LIN {X 0,Y 368.058,Z 315.59,A -85,B 0,C 180,E1 -13017.849,E2 -13017.849} C_VEL
LIN {X 0,Y 375.549,Z 331.898,A -85,B 0,C 180,E1 -13019.02,E2 -13019.02} C_VEL
LIN {X 0,Y 376.727,Z 335.393,A -85,B 0,C 180,E1 -13019.219,E2 -13019.219} C_VEL
LIN {X 0,Y 381.091,Z 359.299,A -85,B 0,C 180,E1 -13020.193,E2 -13020.193} C_VEL
LIN {X 0,Y 377.486,Z 482.299,A -85,B 0,C 180,E1 -13022.675,E2 -13022.675} C_VEL
LIN {X 0,Y 376.481,Z 498.143,A -85,B 0,C 180,E1 -13023.197,E2 -13023.197} C_VEL
LIN {X 0,Y 375.186,Z 512.324,A -85,B 0,C 180,E1 -13023.862,E2 -13023.862} C_VEL
LIN {X 0,Y 373.616,Z 526.793,A -85,B 0,C 180,E1 -13024.762,E2 -13024.762} C_VEL
LIN {X 0,Y 371.852,Z 540.842,A -85,B 0,C 180,E1 -13025.877,E2 -13025.877} C_VEL
LIN {X 0,Y 369.933,Z 554.519,A -85,B 0,C 180,E1 -13027.228,E2 -13027.228} C_VEL
LIN {X 0,Y 367.984,Z 566.938,A -85,B 0,C 180,E1 -13028.724,E2 -13028.724} C_VEL
LIN {X 0,Y 366.187,Z 578.952,A -85,B 0,C 180,E1 -13030.485,E2 -13030.485} C_VEL
LIN {X 0,Y 364.472,Z 589.352,A -85,B 0,C 180,E1 -13032.321,E2 -13032.321} C_VEL
LIN {X 0,Y 363.116,Z 598.534,A -85,B 0,C 180,E1 -13034.279,E2 -13034.279} C_VEL
LIN {X 0,Y 361.947,Z 607.188,A -85,B 0,C 180,E1 -13036.527,E2 -13036.527} C_VEL
LIN {X 0,Y 361.137,Z 614.142,A -85,B 0,C 180,E1 -13038.779,E2 -13038.779} C_VEL
LIN {X 0,Y 360.63,Z 619.607,A -85,B 0,C 180,E1 -13041.031,E2 -13041.031} C_VEL
LIN {X 0,Y 360.378,Z 623.728,A -85,B 0,C 180,E1 -13043.281,E2 -13043.281} C_VEL
LIN {X 0,Y 360.294,Z 626.602,A -85,B 0,C 180,E1 -13045.525,E2 -13045.525} C_VEL
LIN {X 0,Y 360.257,Z 628.286,A -85,B 0,C 180,E1 -13047.764,E2 -13047.764} C_VEL
LIN {X 0,Y 360.36,Z 628.816,A -85,B 0,C 180,E1 -13050,E2 -13050} C_VEL
LIN {X 0,Y 360.258,Z 628.168,A -85,B 0,C 180,E1 -13052.236,E2 -13052.236} C_VEL
LIN {X 0,Y 360.303,Z 626.303,A -85,B 0,C 180,E1 -13054.475,E2 -13054.475} C_VEL
LIN {X 0,Y 360.39,Z 623.235,A -85,B 0,C 180,E1 -13056.72,E2 -13056.72} C_VEL
LIN {X 0,Y 360.63,Z 618.892,A -85,B 0,C 180,E1 -13058.97,E2 -13058.97} C_VEL
LIN {X 0,Y 361.121,Z 613.159,A -85,B 0,C 180,E1 -13061.223,E2 -13061.223} C_VEL
LIN {X 0,Y 361.886,Z 605.883,A -85,B 0,C 180,E1 -13063.477,E2 -13063.477} C_VEL
LIN {X 0,Y 362.881,Z 598.091,A -85,B 0,C 180,E1 -13065.444,E2 -13065.444} C_VEL
LIN {X 0,Y 364.086,Z 588.704,A -85,B 0,C 180,E1 -13067.41,E2 -13067.41} C_VEL
LIN {X 0,Y 365.622,Z 579.166,A -85,B 0,C 180,E1 -13069.073,E2 -13069.073} C_VEL
LIN {X 0,Y 367.142,Z 567.807,A -85,B 0,C 180,E1 -13070.74,E2 -13070.74} C_VEL
LIN {X 0,Y 368.887,Z 555.341,A -85,B 0,C 180,E1 -13072.25,E2 -13072.25} C_VEL
LIN {X 0,Y 370.709,Z 541.567,A -85,B 0,C 180,E1 -13073.609,E2 -13073.609} C_VEL
LIN {X 0,Y 372.318,Z 527.661,A -85,B 0,C 180,E1 -13074.715,E2 -13074.715} C_VEL
LIN {X 0,Y 373.734,Z 513.103,A -85,B 0,C 180,E1 -13075.627,E2 -13075.627} C_VEL
LIN {X 0,Y 374.965,Z 498.276,A -85,B 0,C 180,E1 -13076.32,E2 -13076.32} C_VEL
LIN {X 0,Y 375.87,Z 483.105,A -85,B 0,C 180,E1 -13076.813,E2 -13076.813} C_VEL
LIN {X 0,Y 379.156,Z 359.876,A -85,B 0,C 180,E1 -13079.264,E2 -13079.264} C_VEL
LIN {X 0,Y 375.008,Z 336.566,A -85,B 0,C 180,E1 -13080.111,E2 -13080.111} C_VEL
LIN {X 0,Y 373.504,Z 329.82,A -85,B 0,C 180,E1 -13080.387,E2 -13080.387} C_VEL
LIN {X 0,Y 367.901,Z 316.548,A -85,B 0,C 180,E1 -13081.181,E2 -13081.181} C_VEL
LIN {X 0,Y 364.425,Z 302.708,A -85,B 0,C 180,E1 -13084.338,E2 -13084.338} C_VEL
LIN {X 0,Y 361.869,Z 293.039,A -85,B 0,C 180,E1 -13086.669,E2 -13086.669} C_VEL
LIN {X 0,Y 361.814,Z 293.041,A -85,B 0,C 180,E1 -13089.866,E2 -13089.866} C_VEL
LIN {X 0,Y 361.83,Z 293.034,A -85,B 0,C 180,E1 -13092.829,E2 -13092.829} C_VEL
LIN {X 0,Y 361.814,Z 293.038,A -85,B 0,C 180,E1 -13095.947,E2 -13095.947} C_VEL
LIN {X 0,Y 361.811,Z 293.045,A -85,B 0,C 180,E1 -13099.248,E2 -13099.248} C_VEL
LIN {X 0,Y 361.861,Z 293.038,A -85,B 0,C 180,E1 -13102.98,E2 -13102.98} C_VEL
LIN {X 0,Y 361.858,Z 293.031,A -85,B 0,C 180,E1 -13106.63,E2 -13106.63} C_VEL
LIN {X 0,Y 361.855,Z 293.034,A -85,B 0,C 180,E1 -13109.669,E2 -13109.669} C_VEL
LIN {X 0,Y 361.854,Z 293.033,A -85,B 0,C 180,E1 -13113.466,E2 -13113.466} C_VEL
LIN {X 0,Y 361.86,Z 293.033,A -85,B 0,C 180,E1 -13117.141,E2 -13117.141} C_VEL
LIN {X 0,Y 361.881,Z 293.029,A -85,B 0,C 180,E1 -13120.72,E2 -13120.72} C_VEL
LIN {X 0,Y 361.94,Z 293.021,A -85,B 0,C 180,E1 -13124.224,E2 -13124.224} C_VEL
LIN {X 0,Y 361.995,Z 292.994,A -85,B 0,C 180,E1 -13126.526,E2 -13126.526} C_VEL
LIN {X 0,Y 361.989,Z 293.011,A -85,B 0,C 180,E1 -13129.935,E2 -13129.935} C_VEL
LIN {X 0,Y 362.113,Z 293.004,A -85,B 0,C 180,E1 -13133.311,E2 -13133.311} C_VEL
LIN {X 0,Y 362.248,Z 292.963,A -85,B 0,C 180,E1 -13137.774,E2 -13137.774} C_VEL
LIN {X 0,Y 362.26,Z 292.982,A -85,B 0,C 180,E1 -13142.222,E2 -13142.222} C_VEL
LIN {X 0,Y 362.088,Z 292.973,A -85,B 0,C 180,E1 -13146.686,E2 -13146.686} C_VEL
LIN {X 0,Y 361.967,Z 293.018,A -85,B 0,C 180,E1 -13150.062,E2 -13150.062} C_VEL
LIN {X 0,Y 361.99,Z 293.01,A -85,B 0,C 180,E1 -13153.897,E2 -13153.897} C_VEL
LIN {X 0,Y 361.911,Z 293.004,A -85,B 0,C 180,E1 -13157.913,E2 -13157.913} C_VEL
LIN {X 0,Y 361.851,Z 293.036,A -85,B 0,C 180,E1 -13161.653,E2 -13161.653} C_VEL
LIN {X 0,Y 361.849,Z 293.018,A -85,B 0,C 180,E1 -13165.293,E2 -13165.293} C_VEL
LIN {X 0,Y 361.844,Z 293.02,A -85,B 0,C 180,E1 -13169.072,E2 -13169.072} C_VEL
LIN {X 0,Y 361.835,Z 293.04,A -85,B 0,C 180,E1 -13172.943,E2 -13172.943} C_VEL
LIN {X 0,Y 361.851,Z 293.014,A -85,B 0,C 180,E1 -13175.636,E2 -13175.636} C_VEL
LIN {X 0,Y 361.812,Z 293.032,A -85,B 0,C 180,E1 -13179.016,E2 -13179.016} C_VEL
LIN {X 0,Y 361.817,Z 293.038,A -85,B 0,C 180,E1 -13182.828,E2 -13182.828} C_VEL
LIN {X 0,Y 361.801,Z 293.025,A -85,B 0,C 180,E1 -13185.946,E2 -13185.946} C_VEL
LIN {X 0,Y 361.819,Z 293.044,A -85,B 0,C 180,E1 -13189.244,E2 -13189.244} C_VEL
LIN {X 0,Y 361.847,Z 293.022,A -85,B 0,C 180,E1 -13192.776,E2 -13192.776} C_VEL
LIN {X 0,Y 361.838,Z 293.037,A -85,B 0,C 180,E1 -13195.718,E2 -13195.718} C_VEL
LIN {X 0,Y 361.848,Z 293.022,A -85,B 0,C 180,E1 -13199.67,E2 -13199.67} C_VEL
LIN {X 0,Y 361.937,Z 293.021,A -85,B 0,C 180,E1 -13203.474,E2 -13203.474} C_VEL
LIN {X 0,Y 361.862,Z 293.038,A -85,B 0,C 180,E1 -13207.143,E2 -13207.143} C_VEL
LIN {X 0,Y 361.887,Z 293.03,A -85,B 0,C 180,E1 -13210.722,E2 -13210.722} C_VEL
LIN {X 0,Y 361.916,Z 293.022,A -85,B 0,C 180,E1 -13213.065,E2 -13213.065} C_VEL
LIN {X 0,Y 361.983,Z 293.016,A -85,B 0,C 180,E1 -13216.527,E2 -13216.527} C_VEL
LIN {X 0,Y 362.019,Z 293.011,A -85,B 0,C 180,E1 -13219.937,E2 -13219.937} C_VEL
LIN {X 0,Y 362.143,Z 293,A -85,B 0,C 180,E1 -13223.313,E2 -13223.313} C_VEL
LIN {X 0,Y 362.157,Z 293.106,A -85,B 0,C 180,E1 -13227.149,E2 -13227.149} C_VEL
LIN {X 0,Y 363.617,Z 298.613,A -85,B 0,C 180,E1 -13228.529,E2 -13228.529} C_VEL
LIN {X 0,Y 371.475,Z 315.48,A -85,B 0,C 180,E1 -13229.606,E2 -13229.606} C_VEL
LIN {X 0,Y 379.521,Z 334.569,A -85,B 0,C 180,E1 -13230.695,E2 -13230.695} C_VEL
LIN {X 0,Y 376.136,Z 463.946,A -85,B 0,C 180,E1 -13233.28,E2 -13233.28} C_VEL
LIN {X 0,Y 375.287,Z 479.542,A -85,B 0,C 180,E1 -13233.808,E2 -13233.808} C_VEL
LIN {X 0,Y 374.198,Z 494.266,A -85,B 0,C 180,E1 -13234.523,E2 -13234.523} C_VEL
LIN {X 0,Y 372.901,Z 508.127,A -85,B 0,C 180,E1 -13235.407,E2 -13235.407} C_VEL
LIN {X 0,Y 371.4,Z 521.913,A -85,B 0,C 180,E1 -13236.519,E2 -13236.519} C_VEL
LIN {X 0,Y 369.769,Z 534.735,A -85,B 0,C 180,E1 -13237.791,E2 -13237.791} C_VEL
LIN {X 0,Y 368.026,Z 547.541,A -85,B 0,C 180,E1 -13239.341,E2 -13239.341} C_VEL
LIN {X 0,Y 366.368,Z 559.211,A -85,B 0,C 180,E1 -13241.059,E2 -13241.059} C_VEL
LIN {X 0,Y 364.907,Z 569.028,A -85,B 0,C 180,E1 -13242.796,E2 -13242.796} C_VEL
LIN {X 0,Y 363.601,Z 577.714,A -85,B 0,C 180,E1 -13244.631,E2 -13244.631} C_VEL
LIN {X 0,Y 362.539,Z 581.007,A -85,B 0,C 180,E1 -13245.386,E2 -13245.386} C_VEL
LIN {X 0,Y 359.022,Z 586.056,A -85,B 0,C 180,E1 -13246.622,E2 -13246.622} C_VEL
LIN {X 0,Y 355.55,Z 590.691,A -85,B 0,C 180,E1 -13247.923,E2 -13247.923} C_VEL
LIN {X 0,Y 354.58,Z 593.183,A -85,B 0,C 180,E1 -13248.771,E2 -13248.771} C_VEL
LIN {X 0,Y 353.912,Z 598.756,A -85,B 0,C 180,E1 -13251.048,E2 -13251.048} C_VEL
LIN {X 0,Y 353.485,Z 603.139,A -85,B 0,C 180,E1 -13253.43,E2 -13253.43} C_VEL
LIN {X 0,Y 353.113,Z 606.327,A -85,B 0,C 180,E1 -13255.967,E2 -13255.967} C_VEL
LIN {X 0,Y 352.966,Z 608.076,A -85,B 0,C 180,E1 -13258.545,E2 -13258.545} C_VEL
LIN {X 0,Y 352.946,Z 608.355,A -85,B 0,C 180,E1 -13261.178,E2 -13261.178} C_VEL
LIN {X 0,Y 353.067,Z 607.478,A -85,B 0,C 180,E1 -13263.281,E2 -13263.281} C_VEL
LIN {X 0,Y 353.291,Z 605.694,A -85,B 0,C 180,E1 -13265.357,E2 -13265.357} C_VEL
LIN {X 0,Y 353.628,Z 602.982,A -85,B 0,C 180,E1 -13267.353,E2 -13267.353} C_VEL
LIN {X 0,Y 354.109,Z 599.207,A -85,B 0,C 180,E1 -13269.426,E2 -13269.426} C_VEL
LIN {X 0,Y 354.844,Z 593.89,A -85,B 0,C 180,E1 -13271.671,E2 -13271.671} C_VEL
LIN {X 0,Y 355.764,Z 587.739,A -85,B 0,C 180,E1 -13273.74,E2 -13273.74} C_VEL
LIN {X 0,Y 357.022,Z 579.955,A -85,B 0,C 180,E1 -13275.862,E2 -13275.862} C_VEL
LIN {X 0,Y 358.473,Z 571.612,A -85,B 0,C 180,E1 -13277.738,E2 -13277.738} C_VEL
LIN {X 0,Y 360.098,Z 561.939,A -85,B 0,C 180,E1 -13279.564,E2 -13279.564} C_VEL
LIN {X 0,Y 362.065,Z 550.698,A -85,B 0,C 180,E1 -13281.321,E2 -13281.321} C_VEL
LIN {X 0,Y 364.021,Z 538.332,A -85,B 0,C 180,E1 -13282.921,E2 -13282.921} C_VEL
LIN {X 0,Y 365.86,Z 525.886,A -85,B 0,C 180,E1 -13284.244,E2 -13284.244} C_VEL
LIN {X 0,Y 367.619,Z 512.457,A -85,B 0,C 180,E1 -13285.409,E2 -13285.409} C_VEL
LIN {X 0,Y 369.21,Z 497.84,A -85,B 0,C 180,E1 -13286.415,E2 -13286.415} C_VEL
LIN {X 0,Y 370.537,Z 482.417,A -85,B 0,C 180,E1 -13287.219,E2 -13287.219} C_VEL
LIN {X 0,Y 371.515,Z 467.383,A -85,B 0,C 180,E1 -13287.771,E2 -13287.771} C_VEL
LIN {X 0,Y 372.368,Z 444.646,A -85,B 0,C 180,E1 -13288.285,E2 -13288.285} C_VEL
LIN {X 0,Y 375.579,Z 338.393,A -85,B 0,C 180,E1 -13290.46,E2 -13290.46} C_VEL
LIN {X 0,Y 368.813,Z 323.387,A -85,B 0,C 180,E1 -13291.514,E2 -13291.514} C_VEL
LIN {X 0,Y 361.105,Z 308.12,A -85,B 0,C 180,E1 -13292.747,E2 -13292.747} C_VEL
LIN {X 0,Y 356.555,Z 299.878,A -85,B 0,C 180,E1 -13293.518,E2 -13293.518} C_VEL
LIN {X 0,Y 354.833,Z 293.907,A -85,B 0,C 180,E1 -13295.346,E2 -13295.346} C_VEL
LIN {X 0,Y 354.826,Z 293.917,A -85,B 0,C 180,E1 -13299.116,E2 -13299.116} C_VEL
LIN {X 0,Y 354.885,Z 293.909,A -85,B 0,C 180,E1 -13302.722,E2 -13302.722} C_VEL
LIN {X 0,Y 354.938,Z 293.898,A -85,B 0,C 180,E1 -13306.257,E2 -13306.257} C_VEL
LIN {X 0,Y 354.965,Z 293.894,A -85,B 0,C 180,E1 -13309.738,E2 -13309.738} C_VEL
LIN {X 0,Y 355.114,Z 293.875,A -85,B 0,C 180,E1 -13313.182,E2 -13313.182} C_VEL
LIN {X 0,Y 355.232,Z 293.861,A -85,B 0,C 180,E1 -13317.734,E2 -13317.734} C_VEL
LIN {X 0,Y 355.386,Z 293.84,A -85,B 0,C 180,E1 -13320.002,E2 -13320.002} C_VEL
LIN {X 0,Y 355.231,Z 293.855,A -85,B 0,C 180,E1 -13322.27,E2 -13322.27} C_VEL
LIN {X 0,Y 355.096,Z 293.878,A -85,B 0,C 180,E1 -13326.822,E2 -13326.822} C_VEL
LIN {X 0,Y 354.947,Z 293.896,A -85,B 0,C 180,E1 -13330.267,E2 -13330.267} C_VEL
LIN {X 0,Y 354.935,Z 293.892,A -85,B 0,C 180,E1 -13334.02,E2 -13334.02} C_VEL
LIN {X 0,Y 354.883,Z 293.902,A -85,B 0,C 180,E1 -13338.094,E2 -13338.094} C_VEL
LIN {X 0,Y 354.807,Z 293.915,A -85,B 0,C 180,E1 -13342.109,E2 -13342.109} C_VEL
LIN {X 0,Y 354.799,Z 293.91,A -85,B 0,C 180,E1 -13345.837,E2 -13345.837} C_VEL
LIN {X 0,Y 354.788,Z 293.912,A -85,B 0,C 180,E1 -13349.686,E2 -13349.686} C_VEL
LIN {X 0,Y 354.803,Z 293.912,A -85,B 0,C 180,E1 -13353.704,E2 -13353.704} C_VEL
LIN {X 0,Y 354.787,Z 293.912,A -85,B 0,C 180,E1 -13356.462,E2 -13356.462} C_VEL
LIN {X 0,Y 354.765,Z 293.913,A -85,B 0,C 180,E1 -13359.414,E2 -13359.414} C_VEL
LIN {X 0,Y 354.778,Z 293.917,A -85,B 0,C 180,E1 -13362.867,E2 -13362.867} C_VEL
LIN {X 0,Y 354.759,Z 293.919,A -85,B 0,C 180,E1 -13366.104,E2 -13366.104} C_VEL
LIN {X 0,Y 354.761,Z 293.919,A -85,B 0,C 180,E1 -13369.177,E2 -13369.177} C_VEL
LIN {X 0,Y 354.804,Z 293.968,A -85,B 0,C 180,E1 -13371.351,E2 -13371.351} C_VEL
LIN {X 0,Y 358.32,Z 305.873,A -85,B 0,C 180,E1 -13374.65,E2 -13374.65} C_VEL
LIN {X 0,Y 360.766,Z 315.337,A -85,B 0,C 180,E1 -13377.034,E2 -13377.034} C_VEL
LIN {X 0,Y 368.482,Z 331.416,A -85,B 0,C 180,E1 -13378.283,E2 -13378.283} C_VEL
LIN {X 0,Y 370.94,Z 337.646,A -85,B 0,C 180,E1 -13378.692,E2 -13378.692} C_VEL
LIN {X 0,Y 374.977,Z 360.038,A -85,B 0,C 180,E1 -13379.627,E2 -13379.627} C_VEL
LIN {X 0,Y 371.813,Z 468.07,A -85,B 0,C 180,E1 -13381.84,E2 -13381.84} C_VEL
LIN {X 0,Y 371.035,Z 486.521,A -85,B 0,C 180,E1 -13382.275,E2 -13382.275} C_VEL
LIN {X 0,Y 369.919,Z 501.647,A -85,B 0,C 180,E1 -13382.836,E2 -13382.836} C_VEL
LIN {X 0,Y 368.588,Z 515.054,A -85,B 0,C 180,E1 -13383.517,E2 -13383.517} C_VEL
LIN {X 0,Y 366.949,Z 529.055,A -85,B 0,C 180,E1 -13384.442,E2 -13384.442} C_VEL
LIN {X 0,Y 365.185,Z 542.454,A -85,B 0,C 180,E1 -13385.559,E2 -13385.559} C_VEL
LIN {X 0,Y 363.175,Z 555.788,A -85,B 0,C 180,E1 -13386.93,E2 -13386.93} C_VEL
LIN {X 0,Y 361.346,Z 566.974,A -85,B 0,C 180,E1 -13388.314,E2 -13388.314} C_VEL
LIN {X 0,Y 359.69,Z 577.213,A -85,B 0,C 180,E1 -13389.831,E2 -13389.831} C_VEL
LIN {X 0,Y 357.926,Z 587.792,A -85,B 0,C 180,E1 -13391.69,E2 -13391.69} C_VEL
LIN {X 0,Y 356.429,Z 597.194,A -85,B 0,C 180,E1 -13393.682,E2 -13393.682} C_VEL
LIN {X 0,Y 355.095,Z 605.769,A -85,B 0,C 180,E1 -13395.887,E2 -13395.887} C_VEL
LIN {X 0,Y 354.329,Z 612.377,A -85,B 0,C 180,E1 -13397.98,E2 -13397.98} C_VEL
LIN {X 0,Y 353.653,Z 618.194,A -85,B 0,C 180,E1 -13400.276,E2 -13400.276} C_VEL
LIN {X 0,Y 353.43,Z 621.676,A -85,B 0,C 180,E1 -13401.999,E2 -13401.999} C_VEL
LIN {X 0,Y 353.245,Z 625.147,A -85,B 0,C 180,E1 -13404.291,E2 -13404.291} C_VEL
LIN {X 0,Y 353.194,Z 627.404,A -85,B 0,C 180,E1 -13406.578,E2 -13406.578} C_VEL
LIN {X 0,Y 353.215,Z 628.495,A -85,B 0,C 180,E1 -13408.86,E2 -13408.86} C_VEL
LIN {X 0,Y 353.216,Z 628.432,A -85,B 0,C 180,E1 -13411.141,E2 -13411.141} C_VEL
LIN {X 0,Y 353.196,Z 627.161,A -85,B 0,C 180,E1 -13413.423,E2 -13413.423} C_VEL
LIN {X 0,Y 353.281,Z 624.429,A -85,B 0,C 180,E1 -13415.908,E2 -13415.908} C_VEL
LIN {X 0,Y 353.434,Z 620.972,A -85,B 0,C 180,E1 -13418.002,E2 -13418.002} C_VEL
LIN {X 0,Y 353.735,Z 615.924,A -85,B 0,C 180,E1 -13420.301,E2 -13420.301} C_VEL
LIN {X 0,Y 354.463,Z 609.417,A -85,B 0,C 180,E1 -13422.598,E2 -13422.598} C_VEL
LIN {X 0,Y 355.433,Z 601.258,A -85,B 0,C 180,E1 -13424.895,E2 -13424.895} C_VEL
LIN {X 0,Y 356.637,Z 592.549,A -85,B 0,C 180,E1 -13426.898,E2 -13426.898} C_VEL
LIN {X 0,Y 358.038,Z 583.712,A -85,B 0,C 180,E1 -13428.601,E2 -13428.601} C_VEL
LIN {X 0,Y 359.661,Z 572.424,A -85,B 0,C 180,E1 -13430.423,E2 -13430.423} C_VEL
LIN {X 0,Y 361.345,Z 560.758,A -85,B 0,C 180,E1 -13431.987,E2 -13431.987} C_VEL
LIN {X 0,Y 363.179,Z 548.227,A -85,B 0,C 180,E1 -13433.372,E2 -13433.372} C_VEL
LIN {X 0,Y 364.9,Z 534.489,A -85,B 0,C 180,E1 -13434.614,E2 -13434.614} C_VEL
LIN {X 0,Y 366.507,Z 520.453,A -85,B 0,C 180,E1 -13435.623,E2 -13435.623} C_VEL
LIN {X 0,Y 367.864,Z 505.647,A -85,B 0,C 180,E1 -13436.448,E2 -13436.448} C_VEL
LIN {X 0,Y 369.006,Z 490.703,A -85,B 0,C 180,E1 -13437.047,E2 -13437.047} C_VEL
LIN {X 0,Y 369.726,Z 475.444,A -85,B 0,C 180,E1 -13437.449,E2 -13437.449} C_VEL
LIN {X 0,Y 372.743,Z 359.835,A -85,B 0,C 180,E1 -13439.775,E2 -13439.775} C_VEL
LIN {X 0,Y 367.852,Z 333.219,A -85,B 0,C 180,E1 -13440.787,E2 -13440.787} C_VEL
LIN {X 0,Y 360.608,Z 316.362,A -85,B 0,C 180,E1 -13441.826,E2 -13441.826} C_VEL
LIN {X 0,Y 357.106,Z 302.447,A -85,B 0,C 180,E1 -13445.089,E2 -13445.089} C_VEL
LIN {X 0,Y 354.814,Z 293.918,A -85,B 0,C 180,E1 -13447.219,E2 -13447.219} C_VEL
LIN {X 0,Y 354.765,Z 293.915,A -85,B 0,C 180,E1 -13450.824,E2 -13450.824} C_VEL
LIN {X 0,Y 354.763,Z 293.914,A -85,B 0,C 180,E1 -13453.896,E2 -13453.896} C_VEL
LIN {X 0,Y 354.783,Z 293.917,A -85,B 0,C 180,E1 -13457.659,E2 -13457.659} C_VEL
LIN {X 0,Y 354.787,Z 293.909,A -85,B 0,C 180,E1 -13460.661,E2 -13460.661} C_VEL
LIN {X 0,Y 354.818,Z 293.908,A -85,B 0,C 180,E1 -13464.301,E2 -13464.301} C_VEL
LIN {X 0,Y 354.787,Z 293.915,A -85,B 0,C 180,E1 -13467.665,E2 -13467.665} C_VEL
LIN {X 0,Y 354.796,Z 293.918,A -85,B 0,C 180,E1 -13471.613,E2 -13471.613} C_VEL
LIN {X 0,Y 354.804,Z 293.918,A -85,B 0,C 180,E1 -13475.418,E2 -13475.418} C_VEL
LIN {X 0,Y 354.823,Z 293.915,A -85,B 0,C 180,E1 -13479.111,E2 -13479.111} C_VEL
LIN {X 0,Y 354.878,Z 293.906,A -85,B 0,C 180,E1 -13482.717,E2 -13482.717} C_VEL
LIN {X 0,Y 354.948,Z 293.872,A -85,B 0,C 180,E1 -13486.253,E2 -13486.253} C_VEL
LIN {X 0,Y 354.946,Z 293.885,A -85,B 0,C 180,E1 -13489.733,E2 -13489.733} C_VEL
LIN {X 0,Y 355.079,Z 293.879,A -85,B 0,C 180,E1 -13493.178,E2 -13493.178} C_VEL
LIN {X 0,Y 355.21,Z 293.839,A -85,B 0,C 180,E1 -13497.73,E2 -13497.73} C_VEL
LIN {X 0,Y 355.138,Z 293.871,A -85,B 0,C 180,E1 -13501.132,E2 -13501.132} C_VEL
LIN {X 0,Y 355.222,Z 293.859,A -85,B 0,C 180,E1 -13502.266,E2 -13502.266} C_VEL
LIN {X 0,Y 355.057,Z 293.848,A -85,B 0,C 180,E1 -13506.819,E2 -13506.819} C_VEL
LIN {X 0,Y 354.93,Z 293.894,A -85,B 0,C 180,E1 -13510.263,E2 -13510.263} C_VEL
LIN {X 0,Y 354.934,Z 293.888,A -85,B 0,C 180,E1 -13514.016,E2 -13514.016} C_VEL
LIN {X 0,Y 354.881,Z 293.881,A -85,B 0,C 180,E1 -13518.09,E2 -13518.09} C_VEL
LIN {X 0,Y 354.804,Z 293.912,A -85,B 0,C 180,E1 -13522.106,E2 -13522.106} C_VEL
LIN {X 0,Y 354.788,Z 293.892,A -85,B 0,C 180,E1 -13525.833,E2 -13525.833} C_VEL
LIN {X 0,Y 354.785,Z 293.909,A -85,B 0,C 180,E1 -13529.682,E2 -13529.682} C_VEL
LIN {X 0,Y 354.774,Z 293.916,A -85,B 0,C 180,E1 -13532.332,E2 -13532.332} C_VEL
LIN {X 0,Y 354.805,Z 293.891,A -85,B 0,C 180,E1 -13535.696,E2 -13535.696} C_VEL
LIN {X 0,Y 354.755,Z 293.916,A -85,B 0,C 180,E1 -13539.411,E2 -13539.411} C_VEL
LIN {X 0,Y 354.77,Z 293.915,A -85,B 0,C 180,E1 -13542.865,E2 -13542.865} C_VEL
LIN {X 0,Y 354.75,Z 293.904,A -85,B 0,C 180,E1 -13546.102,E2 -13546.102} C_VEL
LIN {X 0,Y 354.772,Z 293.922,A -85,B 0,C 180,E1 -13549.177,E2 -13549.177} C_VEL
LIN {X 0,Y 354.791,Z 293.902,A -85,B 0,C 180,E1 -13552.401,E2 -13552.401} C_VEL
LIN {X 0,Y 354.796,Z 293.911,A -85,B 0,C 180,E1 -13554.939,E2 -13554.939} C_VEL
LIN {X 0,Y 354.777,Z 293.911,A -85,B 0,C 180,E1 -13558.404,E2 -13558.404} C_VEL
LIN {X 0,Y 354.83,Z 293.909,A -85,B 0,C 180,E1 -13561.617,E2 -13561.617} C_VEL
LIN {X 0,Y 354.882,Z 293.899,A -85,B 0,C 180,E1 -13564.171,E2 -13564.171} C_VEL
LIN {X 0,Y 354.808,Z 293.914,A -85,B 0,C 180,E1 -13567.892,E2 -13567.892} C_VEL
LIN {X 0,Y 354.906,Z 293.902,A -85,B 0,C 180,E1 -13571.891,E2 -13571.891} C_VEL
LIN {X 0,Y 354.926,Z 293.898,A -85,B 0,C 180,E1 -13575.98,E2 -13575.98} C_VEL
LIN {X 0,Y 354.966,Z 293.889,A -85,B 0,C 180,E1 -13579.735,E2 -13579.735} C_VEL
LIN {X 0,Y 355.108,Z 293.878,A -85,B 0,C 180,E1 -13583.18,E2 -13583.18} C_VEL
LIN {X 0,Y 355.014,Z 294.026,A -85,B 0,C 180,E1 -13586.63,E2 -13586.63} C_VEL
LIN {X 0,Y 356.462,Z 298.819,A -85,B 0,C 180,E1 -13587.88,E2 -13587.88} C_VEL
LIN {X 0,Y 364.36,Z 315.598,A -85,B 0,C 180,E1 -13588.992,E2 -13588.992} C_VEL
LIN {X 0,Y 373.116,Z 336.396,A -85,B 0,C 180,E1 -13590.215,E2 -13590.215} C_VEL
LIN {X 0,Y 371.023,Z 416.581,A -85,B 0,C 180,E1 -13591.831,E2 -13591.831} C_VEL
LIN {X 0,Y 369.705,Z 464.398,A -85,B 0,C 180,E1 -13592.826,E2 -13592.826} C_VEL
LIN {X 0,Y 368.795,Z 479.957,A -85,B 0,C 180,E1 -13593.362,E2 -13593.362} C_VEL
LIN {X 0,Y 367.648,Z 494.971,A -85,B 0,C 180,E1 -13594.11,E2 -13594.11} C_VEL
LIN {X 0,Y 366.359,Z 508.325,A -85,B 0,C 180,E1 -13594.978,E2 -13594.978} C_VEL
LIN {X 0,Y 364.857,Z 521.786,A -85,B 0,C 180,E1 -13596.081,E2 -13596.081} C_VEL
LIN {X 0,Y 363.173,Z 534.58,A -85,B 0,C 180,E1 -13597.365,E2 -13597.365} C_VEL
LIN {X 0,Y 361.546,Z 545.82,A -85,B 0,C 180,E1 -13598.726,E2 -13598.726} C_VEL
LIN {X 0,Y 359.857,Z 557.396,A -85,B 0,C 180,E1 -13600.407,E2 -13600.407} C_VEL
LIN {X 0,Y 358.272,Z 567.805,A -85,B 0,C 180,E1 -13602.225,E2 -13602.225} C_VEL
LIN {X 0,Y 356.75,Z 577.441,A -85,B 0,C 180,E1 -13604.255,E2 -13604.255} C_VEL
LIN {X 0,Y 355.564,Z 585.627,A -85,B 0,C 180,E1 -13606.359,E2 -13606.359} C_VEL
LIN {X 0,Y 354.675,Z 592.37,A -85,B 0,C 180,E1 -13608.483,E2 -13608.483} C_VEL
LIN {X 0,Y 354.58,Z 593.183,A -85,B 0,C 180,E1 -13608.771,E2 -13608.771} C_VEL
LIN {X 0,Y 353.655,Z 595.55,A -85,B 0,C 180,E1 -13609.634,E2 -13609.634} C_VEL
LIN {X 0,Y 350.411,Z 599.026,A -85,B 0,C 180,E1 -13611.05,E2 -13611.05} C_VEL
LIN {X 0,Y 347.724,Z 601.447,A -85,B 0,C 180,E1 -13612.219,E2 -13612.219} C_VEL
LIN {X 0,Y 346.51,Z 603.048,A -85,B 0,C 180,E1 -13613.143,E2 -13613.143} C_VEL
LIN {X 0,Y 346.374,Z 603.526,A -85,B 0,C 180,E1 -13613.459,E2 -13613.459} C_VEL
LIN {X 0,Y 346.103,Z 605.868,A -85,B 0,C 180,E1 -13615.24,E2 -13615.24} C_VEL
LIN {X 0,Y 345.876,Z 607.988,A -85,B 0,C 180,E1 -13617.861,E2 -13617.861} C_VEL
LIN {X 0,Y 345.838,Z 608.504,A -85,B 0,C 180,E1 -13619.19,E2 -13619.19} C_VEL
LIN {X 0,Y 345.864,Z 608.538,A -85,B 0,C 180,E1 -13621.417,E2 -13621.417} C_VEL
LIN {X 0,Y 346.01,Z 607.523,A -85,B 0,C 180,E1 -13623.62,E2 -13623.62} C_VEL
LIN {X 0,Y 346.306,Z 605.227,A -85,B 0,C 180,E1 -13626.051,E2 -13626.051} C_VEL
LIN {X 0,Y 346.773,Z 601.988,A -85,B 0,C 180,E1 -13628.28,E2 -13628.28} C_VEL
LIN {X 0,Y 347.309,Z 597.931,A -85,B 0,C 180,E1 -13630.355,E2 -13630.355} C_VEL
LIN {X 0,Y 348.33,Z 591.422,A -85,B 0,C 180,E1 -13632.916,E2 -13632.916} C_VEL
LIN {X 0,Y 349.641,Z 583.667,A -85,B 0,C 180,E1 -13635.293,E2 -13635.293} C_VEL
LIN {X 0,Y 351.107,Z 575.402,A -85,B 0,C 180,E1 -13637.352,E2 -13637.352} C_VEL
LIN {X 0,Y 352.678,Z 566.37,A -85,B 0,C 180,E1 -13639.22,E2 -13639.22} C_VEL
LIN {X 0,Y 354.64,Z 555.663,A -85,B 0,C 180,E1 -13641.06,E2 -13641.06} C_VEL
LIN {X 0,Y 356.776,Z 543.23,A -85,B 0,C 180,E1 -13642.824,E2 -13642.824} C_VEL
LIN {X 0,Y 358.827,Z 530.575,A -85,B 0,C 180,E1 -13644.289,E2 -13644.289} C_VEL
LIN {X 0,Y 360.805,Z 516.621,A -85,B 0,C 180,E1 -13645.609,E2 -13645.609} C_VEL
LIN {X 0,Y 362.651,Z 501.67,A -85,B 0,C 180,E1 -13646.719,E2 -13646.719} C_VEL
LIN {X 0,Y 364.044,Z 486.652,A -85,B 0,C 180,E1 -13647.58,E2 -13647.58} C_VEL
LIN {X 0,Y 365.157,Z 472.085,A -85,B 0,C 180,E1 -13648.182,E2 -13648.182} C_VEL
LIN {X 0,Y 365.897,Z 456.256,A -85,B 0,C 180,E1 -13648.612,E2 -13648.612} C_VEL
LIN {X 0,Y 369.552,Z 340.412,A -85,B 0,C 180,E1 -13651.019,E2 -13651.019} C_VEL
LIN {X 0,Y 362.724,Z 325.243,A -85,B 0,C 180,E1 -13652.128,E2 -13652.128} C_VEL
LIN {X 0,Y 354.898,Z 310.097,A -85,B 0,C 180,E1 -13653.425,E2 -13653.425} C_VEL
LIN {X 0,Y 349.353,Z 300.102,A -85,B 0,C 180,E1 -13654.42,E2 -13654.42} C_VEL
LIN {X 0,Y 347.768,Z 294.793,A -85,B 0,C 180,E1 -13656.163,E2 -13656.163} C_VEL
LIN {X 0,Y 347.8,Z 294.788,A -85,B 0,C 180,E1 -13659.911,E2 -13659.911} C_VEL
LIN {X 0,Y 347.853,Z 294.784,A -85,B 0,C 180,E1 -13662.361,E2 -13662.361} C_VEL
LIN {X 0,Y 347.885,Z 294.777,A -85,B 0,C 180,E1 -13665.973,E2 -13665.973} C_VEL
LIN {X 0,Y 347.916,Z 294.771,A -85,B 0,C 180,E1 -13669.527,E2 -13669.527} C_VEL
LIN {X 0,Y 348.08,Z 294.752,A -85,B 0,C 180,E1 -13673.044,E2 -13673.044} C_VEL
LIN {X 0,Y 348.194,Z 294.738,A -85,B 0,C 180,E1 -13677.688,E2 -13677.688} C_VEL
LIN {X 0,Y 348.335,Z 294.718,A -85,B 0,C 180,E1 -13680.002,E2 -13680.002} C_VEL
LIN {X 0,Y 348.193,Z 294.732,A -85,B 0,C 180,E1 -13682.315,E2 -13682.315} C_VEL
LIN {X 0,Y 348.063,Z 294.752,A -85,B 0,C 180,E1 -13686.96,E2 -13686.96} C_VEL
LIN {X 0,Y 347.887,Z 294.773,A -85,B 0,C 180,E1 -13690.477,E2 -13690.477} C_VEL
LIN {X 0,Y 347.892,Z 294.77,A -85,B 0,C 180,E1 -13694.152,E2 -13694.152} C_VEL
LIN {X 0,Y 347.822,Z 294.783,A -85,B 0,C 180,E1 -13698.261,E2 -13698.261} C_VEL
LIN {X 0,Y 347.76,Z 294.791,A -85,B 0,C 180,E1 -13701.627,E2 -13701.627} C_VEL
LIN {X 0,Y 347.734,Z 294.792,A -85,B 0,C 180,E1 -13705.116,E2 -13705.116} C_VEL
LIN {X 0,Y 347.73,Z 294.794,A -85,B 0,C 180,E1 -13707.702,E2 -13707.702} C_VEL
LIN {X 0,Y 347.724,Z 294.797,A -85,B 0,C 180,E1 -13710.352,E2 -13710.352} C_VEL
LIN {X 0,Y 347.744,Z 294.789,A -85,B 0,C 180,E1 -13714.045,E2 -13714.045} C_VEL
LIN {X 0,Y 347.75,Z 294.789,A -85,B 0,C 180,E1 -13717.324,E2 -13717.324} C_VEL
LIN {X 0,Y 347.693,Z 294.802,A -85,B 0,C 180,E1 -13720.304,E2 -13720.304} C_VEL
LIN {X 0,Y 347.718,Z 294.794,A -85,B 0,C 180,E1 -13723.41,E2 -13723.41} C_VEL
LIN {X 0,Y 347.721,Z 294.798,A -85,B 0,C 180,E1 -13726.689,E2 -13726.689} C_VEL
LIN {X 0,Y 347.7,Z 294.803,A -85,B 0,C 180,E1 -13730.184,E2 -13730.184} C_VEL
LIN {X 0,Y 347.754,Z 295.006,A -85,B 0,C 180,E1 -13730.615,E2 -13730.615} C_VEL
LIN {X 0,Y 351.123,Z 305.948,A -85,B 0,C 180,E1 -13733.781,E2 -13733.781} C_VEL
LIN {X 0,Y 353.576,Z 315.15,A -85,B 0,C 180,E1 -13736.184,E2 -13736.184} C_VEL
LIN {X 0,Y 361.809,Z 331.947,A -85,B 0,C 180,E1 -13737.575,E2 -13737.575} C_VEL
LIN {X 0,Y 365.262,Z 340.181,A -85,B 0,C 180,E1 -13738.158,E2 -13738.158} C_VEL
LIN {X 0,Y 368.986,Z 361.202,A -85,B 0,C 180,E1 -13739.061,E2 -13739.061} C_VEL
LIN {X 0,Y 365.624,Z 469.926,A -85,B 0,C 180,E1 -13741.319,E2 -13741.319} C_VEL
LIN {X 0,Y 364.826,Z 487.588,A -85,B 0,C 180,E1 -13741.761,E2 -13741.761} C_VEL
LIN {X 0,Y 363.578,Z 503.011,A -85,B 0,C 180,E1 -13742.361,E2 -13742.361} C_VEL
LIN {X 0,Y 362.154,Z 516.534,A -85,B 0,C 180,E1 -13743.086,E2 -13743.086} C_VEL
LIN {X 0,Y 360.325,Z 531.076,A -85,B 0,C 180,E1 -13744.096,E2 -13744.096} C_VEL
LIN {X 0,Y 358.503,Z 543.999,A -85,B 0,C 180,E1 -13745.228,E2 -13745.228} C_VEL
LIN {X 0,Y 356.423,Z 557.028,A -85,B 0,C 180,E1 -13746.621,E2 -13746.621} C_VEL
LIN {X 0,Y 354.374,Z 568.971,A -85,B 0,C 180,E1 -13748.171,E2 -13748.171} C_VEL
LIN {X 0,Y 352.464,Z 580.506,A -85,B 0,C 180,E1 -13749.99,E2 -13749.99} C_VEL
LIN {X 0,Y 350.602,Z 590.606,A -85,B 0,C 180,E1 -13751.899,E2 -13751.899} C_VEL
LIN {X 0,Y 349.155,Z 599.513,A -85,B 0,C 180,E1 -13753.933,E2 -13753.933} C_VEL
LIN {X 0,Y 347.988,Z 606.956,A -85,B 0,C 180,E1 -13755.975,E2 -13755.975} C_VEL
LIN {X 0,Y 347.133,Z 613.875,A -85,B 0,C 180,E1 -13758.32,E2 -13758.32} C_VEL
LIN {X 0,Y 346.511,Z 619.318,A -85,B 0,C 180,E1 -13760.663,E2 -13760.663} C_VEL
LIN {X 0,Y 346.223,Z 623.408,A -85,B 0,C 180,E1 -13763.005,E2 -13763.005} C_VEL
LIN {X 0,Y 346.094,Z 626.248,A -85,B 0,C 180,E1 -13765.342,E2 -13765.342} C_VEL
LIN {X 0,Y 346.076,Z 627.901,A -85,B 0,C 180,E1 -13767.673,E2 -13767.673} C_VEL
LIN {X 0,Y 346.166,Z 628.4,A -85,B 0,C 180,E1 -13770,E2 -13770} C_VEL
LIN {X 0,Y 346.077,Z 627.731,A -85,B 0,C 180,E1 -13772.328,E2 -13772.328} C_VEL
LIN {X 0,Y 346.118,Z 625.837,A -85,B 0,C 180,E1 -13774.659,E2 -13774.659} C_VEL
LIN {X 0,Y 346.232,Z 622.73,A -85,B 0,C 180,E1 -13776.996,E2 -13776.996} C_VEL
LIN {X 0,Y 346.508,Z 618.342,A -85,B 0,C 180,E1 -13779.338,E2 -13779.338} C_VEL
LIN {X 0,Y 347.078,Z 612.559,A -85,B 0,C 180,E1 -13781.683,E2 -13781.683} C_VEL
LIN {X 0,Y 347.792,Z 606.246,A -85,B 0,C 180,E1 -13783.736,E2 -13783.736} C_VEL
LIN {X 0,Y 348.865,Z 598.613,A -85,B 0,C 180,E1 -13785.781,E2 -13785.781} C_VEL
LIN {X 0,Y 350.177,Z 589.404,A -85,B 0,C 180,E1 -13787.822,E2 -13787.822} C_VEL
LIN {X 0,Y 351.992,Z 578.275,A -85,B 0,C 180,E1 -13789.842,E2 -13789.842} C_VEL
LIN {X 0,Y 353.742,Z 566.826,A -85,B 0,C 180,E1 -13791.565,E2 -13791.565} C_VEL
LIN {X 0,Y 355.47,Z 555.499,A -85,B 0,C 180,E1 -13792.984,E2 -13792.984} C_VEL
LIN {X 0,Y 357.396,Z 541.871,A -85,B 0,C 180,E1 -13794.39,E2 -13794.39} C_VEL
LIN {X 0,Y 359.077,Z 528.48,A -85,B 0,C 180,E1 -13795.505,E2 -13795.505} C_VEL
LIN {X 0,Y 360.556,Z 514.845,A -85,B 0,C 180,E1 -13796.408,E2 -13796.408} C_VEL
LIN {X 0,Y 361.886,Z 500.075,A -85,B 0,C 180,E1 -13797.154,E2 -13797.154} C_VEL
LIN {X 0,Y 362.914,Z 484.814,A -85,B 0,C 180,E1 -13797.695,E2 -13797.695} C_VEL
LIN {X 0,Y 363.825,Z 457.828,A -85,B 0,C 180,E1 -13798.286,E2 -13798.286} C_VEL
LIN {X 0,Y 366.457,Z 360.809,A -85,B 0,C 180,E1 -13800.273,E2 -13800.273} C_VEL
LIN {X 0,Y 361.913,Z 335.952,A -85,B 0,C 180,E1 -13801.238,E2 -13801.238} C_VEL
LIN {X 0,Y 353.315,Z 316.075,A -85,B 0,C 180,E1 -13802.519,E2 -13802.519} C_VEL
LIN {X 0,Y 350.066,Z 303.274,A -85,B 0,C 180,E1 -13805.606,E2 -13805.606} C_VEL
LIN {X 0,Y 347.759,Z 294.792,A -85,B 0,C 180,E1 -13807.805,E2 -13807.805} C_VEL
LIN {X 0,Y 347.742,Z 294.796,A -85,B 0,C 180,E1 -13811.831,E2 -13811.831} C_VEL
LIN {X 0,Y 347.701,Z 294.8,A -85,B 0,C 180,E1 -13815.027,E2 -13815.027} C_VEL
LIN {X 0,Y 347.739,Z 294.801,A -85,B 0,C 180,E1 -13818.399,E2 -13818.399} C_VEL
LIN {X 0,Y 347.762,Z 294.792,A -85,B 0,C 180,E1 -13822.013,E2 -13822.013} C_VEL
LIN {X 0,Y 347.743,Z 294.781,A -85,B 0,C 180,E1 -13825.534,E2 -13825.534} C_VEL
LIN {X 0,Y 347.745,Z 294.793,A -85,B 0,C 180,E1 -13828.299,E2 -13828.299} C_VEL
LIN {X 0,Y 347.744,Z 294.792,A -85,B 0,C 180,E1 -13830.983,E2 -13830.983} C_VEL
LIN {X 0,Y 347.735,Z 294.793,A -85,B 0,C 180,E1 -13833.598,E2 -13833.598} C_VEL
LIN {X 0,Y 347.747,Z 294.792,A -85,B 0,C 180,E1 -13836.157,E2 -13836.157} C_VEL
LIN {X 0,Y 347.796,Z 294.786,A -85,B 0,C 180,E1 -13839.907,E2 -13839.907} C_VEL
LIN {X 0,Y 347.829,Z 294.786,A -85,B 0,C 180,E1 -13843.567,E2 -13843.567} C_VEL
LIN {X 0,Y 347.883,Z 294.746,A -85,B 0,C 180,E1 -13847.159,E2 -13847.159} C_VEL
LIN {X 0,Y 347.929,Z 294.765,A -85,B 0,C 180,E1 -13850.699,E2 -13850.699} C_VEL
LIN {X 0,Y 348.03,Z 294.748,A -85,B 0,C 180,E1 -13854.203,E2 -13854.203} C_VEL
LIN {X 0,Y 348.147,Z 294.717,A -85,B 0,C 180,E1 -13857.684,E2 -13857.684} C_VEL
LIN {X 0,Y 348.109,Z 294.747,A -85,B 0,C 180,E1 -13861.155,E2 -13861.155} C_VEL
LIN {X 0,Y 348.183,Z 294.735,A -85,B 0,C 180,E1 -13862.312,E2 -13862.312} C_VEL
LIN {X 0,Y 348.028,Z 294.724,A -85,B 0,C 180,E1 -13866.957,E2 -13866.957} C_VEL
LIN {X 0,Y 347.873,Z 294.773,A -85,B 0,C 180,E1 -13870.474,E2 -13870.474} C_VEL
LIN {X 0,Y 347.891,Z 294.764,A -85,B 0,C 180,E1 -13874.148,E2 -13874.148} C_VEL
LIN {X 0,Y 347.82,Z 294.762,A -85,B 0,C 180,E1 -13878.257,E2 -13878.257} C_VEL
LIN {X 0,Y 347.758,Z 294.792,A -85,B 0,C 180,E1 -13881.624,E2 -13881.624} C_VEL
LIN {X 0,Y 347.725,Z 294.779,A -85,B 0,C 180,E1 -13885.112,E2 -13885.112} C_VEL
LIN {X 0,Y 347.713,Z 294.769,A -85,B 0,C 180,E1 -13887.7,E2 -13887.7} C_VEL
LIN {X 0,Y 347.727,Z 294.789,A -85,B 0,C 180,E1 -13890.347,E2 -13890.347} C_VEL
LIN {X 0,Y 347.736,Z 294.786,A -85,B 0,C 180,E1 -13894.042,E2 -13894.042} C_VEL
LIN {X 0,Y 347.742,Z 294.769,A -85,B 0,C 180,E1 -13897.32,E2 -13897.32} C_VEL
LIN {X 0,Y 347.727,Z 294.795,A -85,B 0,C 180,E1 -13901.599,E2 -13901.599} C_VEL
LIN {X 0,Y 347.687,Z 294.78,A -85,B 0,C 180,E1 -13905.026,E2 -13905.026} C_VEL
LIN {X 0,Y 347.735,Z 294.793,A -85,B 0,C 180,E1 -13908.396,E2 -13908.396} C_VEL
LIN {X 0,Y 347.758,Z 294.781,A -85,B 0,C 180,E1 -13912.01,E2 -13912.01} C_VEL
LIN {X 0,Y 347.729,Z 294.796,A -85,B 0,C 180,E1 -13915.535,E2 -13915.535} C_VEL
LIN {X 0,Y 347.729,Z 294.79,A -85,B 0,C 180,E1 -13918.299,E2 -13918.299} C_VEL
LIN {X 0,Y 347.762,Z 294.784,A -85,B 0,C 180,E1 -13920.986,E2 -13920.986} C_VEL
LIN {X 0,Y 347.814,Z 294.78,A -85,B 0,C 180,E1 -13923.606,E2 -13923.606} C_VEL
LIN {X 0,Y 347.768,Z 294.786,A -85,B 0,C 180,E1 -13926.16,E2 -13926.16} C_VEL
LIN {X 0,Y 347.788,Z 294.78,A -85,B 0,C 180,E1 -13929.908,E2 -13929.908} C_VEL
LIN {X 0,Y 347.849,Z 294.782,A -85,B 0,C 180,E1 -13932.358,E2 -13932.358} C_VEL
LIN {X 0,Y 347.881,Z 294.776,A -85,B 0,C 180,E1 -13935.97,E2 -13935.97} C_VEL
LIN {X 0,Y 347.916,Z 294.767,A -85,B 0,C 180,E1 -13939.525,E2 -13939.525} C_VEL
LIN {X 0,Y 348.074,Z 294.755,A -85,B 0,C 180,E1 -13943.041,E2 -13943.041} C_VEL
LIN {X 0,Y 347.91,Z 294.926,A -85,B 0,C 180,E1 -13946.09,E2 -13946.09} C_VEL
LIN {X 0,Y 349.241,Z 299.099,A -85,B 0,C 180,E1 -13947.195,E2 -13947.195} C_VEL
LIN {X 0,Y 358.255,Z 318.023,A -85,B 0,C 180,E1 -13948.504,E2 -13948.504} C_VEL
LIN {X 0,Y 365.449,Z 335.005,A -85,B 0,C 180,E1 -13949.536,E2 -13949.536} C_VEL
LIN {X 0,Y 366.923,Z 338.527,A -85,B 0,C 180,E1 -13949.742,E2 -13949.742} C_VEL
LIN {X 0,Y 363.338,Z 463.674,A -85,B 0,C 180,E1 -13952.321,E2 -13952.321} C_VEL
LIN {X 0,Y 362.48,Z 479.055,A -85,B 0,C 180,E1 -13952.847,E2 -13952.847} C_VEL
LIN {X 0,Y 361.357,Z 493.44,A -85,B 0,C 180,E1 -13953.554,E2 -13953.554} C_VEL
LIN {X 0,Y 359.945,Z 507.719,A -85,B 0,C 180,E1 -13954.479,E2 -13954.479} C_VEL
LIN {X 0,Y 358.307,Z 521.682,A -85,B 0,C 180,E1 -13955.628,E2 -13955.628} C_VEL
LIN {X 0,Y 356.569,Z 534.525,A -85,B 0,C 180,E1 -13956.933,E2 -13956.933} C_VEL
LIN {X 0,Y 354.785,Z 546.519,A -85,B 0,C 180,E1 -13958.412,E2 -13958.412} C_VEL
LIN {X 0,Y 353.111,Z 557.425,A -85,B 0,C 180,E1 -13960.029,E2 -13960.029} C_VEL
LIN {X 0,Y 351.505,Z 567.447,A -85,B 0,C 180,E1 -13961.798,E2 -13961.798} C_VEL
LIN {X 0,Y 350.09,Z 576.219,A -85,B 0,C 180,E1 -13963.643,E2 -13963.643} C_VEL
LIN {X 0,Y 348.755,Z 584.67,A -85,B 0,C 180,E1 -13965.785,E2 -13965.785} C_VEL
LIN {X 0,Y 347.707,Z 592.353,A -85,B 0,C 180,E1 -13968.207,E2 -13968.207} C_VEL
LIN {X 0,Y 346.909,Z 598.498,A -85,B 0,C 180,E1 -13970.686,E2 -13970.686} C_VEL
LIN {X 0,Y 346.541,Z 602.311,A -85,B 0,C 180,E1 -13972.663,E2 -13972.663} C_VEL
LIN {X 0,Y 346.374,Z 603.526,A -85,B 0,C 180,E1 -13973.459,E2 -13973.459} C_VEL
LIN {X 0,Y 345.563,Z 604.899,A -85,B 0,C 180,E1 -13974.401,E2 -13974.401} C_VEL
LIN {X 0,Y 342.501,Z 606.758,A -85,B 0,C 180,E1 -13975.941,E2 -13975.941} C_VEL
LIN {X 0,Y 339.957,Z 607.823,A -85,B 0,C 180,E1 -13977.199,E2 -13977.199} C_VEL
LIN {X 0,Y 338.848,Z 608.35,A -85,B 0,C 180,E1 -13978.182,E2 -13978.182} C_VEL
LIN {X 0,Y 338.747,Z 608.468,A -85,B 0,C 180,E1 -13978.516,E2 -13978.516} C_VEL
LIN {X 0,Y 338.771,Z 608.771,A -85,B 0,C 180,E1 -13981.24,E2 -13981.24} C_VEL
LIN {X 0,Y 338.837,Z 608.348,A -85,B 0,C 180,E1 -13982.633,E2 -13982.633} C_VEL
LIN {X 0,Y 338.956,Z 607.524,A -85,B 0,C 180,E1 -13984.042,E2 -13984.042} C_VEL
LIN {X 0,Y 339.232,Z 605.561,A -85,B 0,C 180,E1 -13986.106,E2 -13986.106} C_VEL
LIN {X 0,Y 339.72,Z 602.421,A -85,B 0,C 180,E1 -13988.36,E2 -13988.36} C_VEL
LIN {X 0,Y 340.353,Z 597.979,A -85,B 0,C 180,E1 -13990.686,E2 -13990.686} C_VEL
LIN {X 0,Y 341.196,Z 592.712,A -85,B 0,C 180,E1 -13992.821,E2 -13992.821} C_VEL
LIN {X 0,Y 342.405,Z 585.835,A -85,B 0,C 180,E1 -13995.073,E2 -13995.073} C_VEL
LIN {X 0,Y 344.004,Z 577.261,A -85,B 0,C 180,E1 -13997.346,E2 -13997.346} C_VEL
LIN {X 0,Y 345.785,Z 567.644,A -85,B 0,C 180,E1 -13999.432,E2 -13999.432} C_VEL
LIN {X 0,Y 347.717,Z 557.76,A -85,B 0,C 180,E1 -14001.206,E2 -14001.206} C_VEL
LIN {X 0,Y 349.818,Z 546.201,A -85,B 0,C 180,E1 -14002.939,E2 -14002.939} C_VEL
LIN {X 0,Y 351.949,Z 533.885,A -85,B 0,C 180,E1 -14004.459,E2 -14004.459} C_VEL
LIN {X 0,Y 354.017,Z 520.129,A -85,B 0,C 180,E1 -14005.849,E2 -14005.849} C_VEL
LIN {X 0,Y 355.856,Z 506.278,A -85,B 0,C 180,E1 -14006.965,E2 -14006.965} C_VEL
LIN {X 0,Y 357.409,Z 492.107,A -85,B 0,C 180,E1 -14007.861,E2 -14007.861} C_VEL
LIN {X 0,Y 358.684,Z 477.141,A -85,B 0,C 180,E1 -14008.568,E2 -14008.568} C_VEL
LIN {X 0,Y 359.604,Z 462.211,A -85,B 0,C 180,E1 -14009.049,E2 -14009.049} C_VEL
LIN {X 0,Y 363.624,Z 342.543,A -85,B 0,C 180,E1 -14011.596,E2 -14011.596} C_VEL
LIN {X 0,Y 355.784,Z 325.384,A -85,B 0,C 180,E1 -14012.917,E2 -14012.917} C_VEL
LIN {X 0,Y 348.944,Z 312.377,A -85,B 0,C 180,E1 -14014.103,E2 -14014.103} C_VEL
LIN {X 0,Y 343.62,Z 303.297,A -85,B 0,C 180,E1 -14015.046,E2 -14015.046} C_VEL
LIN {X 0,Y 342.133,Z 300.452,A -85,B 0,C 180,E1 -14015.355,E2 -14015.355} C_VEL
LIN {X 0,Y 340.712,Z 295.672,A -85,B 0,C 180,E1 -14016.929,E2 -14016.929} C_VEL
LIN {X 0,Y 340.778,Z 295.656,A -85,B 0,C 180,E1 -14020.735,E2 -14020.735} C_VEL
LIN {X 0,Y 340.773,Z 295.664,A -85,B 0,C 180,E1 -14023.22,E2 -14023.22} C_VEL
LIN {X 0,Y 340.831,Z 295.654,A -85,B 0,C 180,E1 -14026.892,E2 -14026.892} C_VEL
LIN {X 0,Y 340.902,Z 295.647,A -85,B 0,C 180,E1 -14030.509,E2 -14030.509} C_VEL
LIN {X 0,Y 341.048,Z 295.63,A -85,B 0,C 180,E1 -14032.9,E2 -14032.9} C_VEL
LIN {X 0,Y 341.156,Z 295.615,A -85,B 0,C 180,E1 -14037.641,E2 -14037.641} C_VEL
LIN {X 0,Y 341.285,Z 295.596,A -85,B 0,C 180,E1 -14040.002,E2 -14040.002} C_VEL
LIN {X 0,Y 341.155,Z 295.609,A -85,B 0,C 180,E1 -14042.363,E2 -14042.363} C_VEL
LIN {X 0,Y 341.011,Z 295.629,A -85,B 0,C 180,E1 -14047.105,E2 -14047.105} C_VEL
LIN {X 0,Y 340.839,Z 295.649,A -85,B 0,C 180,E1 -14050.697,E2 -14050.697} C_VEL
LIN {X 0,Y 340.856,Z 295.646,A -85,B 0,C 180,E1 -14054.327,E2 -14054.327} C_VEL
LIN {X 0,Y 340.779,Z 295.662,A -85,B 0,C 180,E1 -14058.442,E2 -14058.442} C_VEL
LIN {X 0,Y 340.712,Z 295.67,A -85,B 0,C 180,E1 -14061.844,E2 -14061.844} C_VEL
LIN {X 0,Y 340.67,Z 295.671,A -85,B 0,C 180,E1 -14065.674,E2 -14065.674} C_VEL
LIN {X 0,Y 340.676,Z 295.67,A -85,B 0,C 180,E1 -14068.327,E2 -14068.327} C_VEL
LIN {X 0,Y 340.678,Z 295.668,A -85,B 0,C 180,E1 -14071.048,E2 -14071.048} C_VEL
LIN {X 0,Y 340.711,Z 295.667,A -85,B 0,C 180,E1 -14075.281,E2 -14075.281} C_VEL
LIN {X 0,Y 340.689,Z 295.67,A -85,B 0,C 180,E1 -14078.384,E2 -14078.384} C_VEL
LIN {X 0,Y 340.687,Z 295.671,A -85,B 0,C 180,E1 -14082.045,E2 -14082.045} C_VEL
LIN {X 0,Y 340.647,Z 295.677,A -85,B 0,C 180,E1 -14086.229,E2 -14086.229} C_VEL
LIN {X 0,Y 340.675,Z 295.716,A -85,B 0,C 180,E1 -14089.733,E2 -14089.733} C_VEL
LIN {X 0,Y 343.834,Z 306.102,A -85,B 0,C 180,E1 -14092.862,E2 -14092.862} C_VEL
LIN {X 0,Y 346.294,Z 314.792,A -85,B 0,C 180,E1 -14095.26,E2 -14095.26} C_VEL
LIN {X 0,Y 355.259,Z 332.796,A -85,B 0,C 180,E1 -14096.849,E2 -14096.849} C_VEL
LIN {X 0,Y 359.651,Z 342.984,A -85,B 0,C 180,E1 -14097.614,E2 -14097.614} C_VEL
LIN {X 0,Y 363.033,Z 362.311,A -85,B 0,C 180,E1 -14098.469,E2 -14098.469} C_VEL
LIN {X 0,Y 359.604,Z 468.389,A -85,B 0,C 180,E1 -14100.713,E2 -14100.713} C_VEL
LIN {X 0,Y 358.778,Z 486.489,A -85,B 0,C 180,E1 -14101.161,E2 -14101.161} C_VEL
LIN {X 0,Y 357.515,Z 501.445,A -85,B 0,C 180,E1 -14101.731,E2 -14101.731} C_VEL
LIN {X 0,Y 355.934,Z 516.112,A -85,B 0,C 180,E1 -14102.514,E2 -14102.514} C_VEL
LIN {X 0,Y 354.091,Z 530.554,A -85,B 0,C 180,E1 -14103.531,E2 -14103.531} C_VEL
LIN {X 0,Y 352.063,Z 544.194,A -85,B 0,C 180,E1 -14104.743,E2 -14104.743} C_VEL
LIN {X 0,Y 349.91,Z 557.128,A -85,B 0,C 180,E1 -14106.159,E2 -14106.159} C_VEL
LIN {X 0,Y 347.76,Z 568.999,A -85,B 0,C 180,E1 -14107.734,E2 -14107.734} C_VEL
LIN {X 0,Y 345.818,Z 580.05,A -85,B 0,C 180,E1 -14109.505,E2 -14109.505} C_VEL
LIN {X 0,Y 344.092,Z 589.193,A -85,B 0,C 180,E1 -14111.236,E2 -14111.236} C_VEL
LIN {X 0,Y 342.478,Z 598.304,A -85,B 0,C 180,E1 -14113.305,E2 -14113.305} C_VEL
LIN {X 0,Y 341.021,Z 606.86,A -85,B 0,C 180,E1 -14115.683,E2 -14115.683} C_VEL
LIN {X 0,Y 340.109,Z 613.753,A -85,B 0,C 180,E1 -14118.075,E2 -14118.075} C_VEL
LIN {X 0,Y 339.439,Z 619.177,A -85,B 0,C 180,E1 -14120.466,E2 -14120.466} C_VEL
LIN {X 0,Y 339.143,Z 623.248,A -85,B 0,C 180,E1 -14122.858,E2 -14122.858} C_VEL
LIN {X 0,Y 339,Z 626.073,A -85,B 0,C 180,E1 -14125.244,E2 -14125.244} C_VEL
LIN {X 0,Y 338.99,Z 627.71,A -85,B 0,C 180,E1 -14127.624,E2 -14127.624} C_VEL
LIN {X 0,Y 339.068,Z 628.191,A -85,B 0,C 180,E1 -14130,E2 -14130} C_VEL
LIN {X 0,Y 338.991,Z 627.508,A -85,B 0,C 180,E1 -14132.377,E2 -14132.377} C_VEL
LIN {X 0,Y 339.023,Z 625.6,A -85,B 0,C 180,E1 -14134.757,E2 -14134.757} C_VEL
LIN {X 0,Y 339.153,Z 622.472,A -85,B 0,C 180,E1 -14137.143,E2 -14137.143} C_VEL
LIN {X 0,Y 339.431,Z 618.06,A -85,B 0,C 180,E1 -14139.535,E2 -14139.535} C_VEL
LIN {X 0,Y 340.06,Z 612.253,A -85,B 0,C 180,E1 -14141.927,E2 -14141.927} C_VEL
LIN {X 0,Y 340.871,Z 604.995,A -85,B 0,C 180,E1 -14144.292,E2 -14144.292} C_VEL
LIN {X 0,Y 342.12,Z 596.998,A -85,B 0,C 180,E1 -14146.407,E2 -14146.407} C_VEL
LIN {X 0,Y 343.616,Z 587.502,A -85,B 0,C 180,E1 -14148.483,E2 -14148.483} C_VEL
LIN {X 0,Y 345.197,Z 577.825,A -85,B 0,C 180,E1 -14150.25,E2 -14150.25} C_VEL
LIN {X 0,Y 346.973,Z 566.309,A -85,B 0,C 180,E1 -14152.007,E2 -14152.007} C_VEL
LIN {X 0,Y 349.07,Z 553.651,A -85,B 0,C 180,E1 -14153.588,E2 -14153.588} C_VEL
LIN {X 0,Y 350.874,Z 541.2,A -85,B 0,C 180,E1 -14154.874,E2 -14154.874} C_VEL
LIN {X 0,Y 352.65,Z 527.72,A -85,B 0,C 180,E1 -14156.004,E2 -14156.004} C_VEL
LIN {X 0,Y 354.11,Z 514.388,A -85,B 0,C 180,E1 -14156.894,E2 -14156.894} C_VEL
LIN {X 0,Y 355.477,Z 499.664,A -85,B 0,C 180,E1 -14157.645,E2 -14157.645} C_VEL
LIN {X 0,Y 356.549,Z 484.301,A -85,B 0,C 180,E1 -14158.193,E2 -14158.193} C_VEL
LIN {X 0,Y 357.627,Z 451.956,A -85,B 0,C 180,E1 -14158.902,E2 -14158.902} C_VEL
LIN {X 0,Y 360.2,Z 362.053,A -85,B 0,C 180,E1 -14160.775,E2 -14160.775} C_VEL
LIN {X 0,Y 355.964,Z 338.648,A -85,B 0,C 180,E1 -14161.703,E2 -14161.703} C_VEL
LIN {X 0,Y 347.593,Z 319.481,A -85,B 0,C 180,E1 -14162.955,E2 -14162.955} C_VEL
LIN {X 0,Y 346.032,Z 315.929,A -85,B 0,C 180,E1 -14163.21,E2 -14163.21} C_VEL
LIN {X 0,Y 342.691,Z 302.704,A -85,B 0,C 180,E1 -14166.494,E2 -14166.494} C_VEL
LIN {X 0,Y 340.706,Z 295.67,A -85,B 0,C 180,E1 -14168.383,E2 -14168.383} C_VEL
LIN {X 0,Y 340.692,Z 295.674,A -85,B 0,C 180,E1 -14172.043,E2 -14172.043} C_VEL
LIN {X 0,Y 340.651,Z 295.672,A -85,B 0,C 180,E1 -14176.227,E2 -14176.227} C_VEL
LIN {X 0,Y 340.67,Z 295.68,A -85,B 0,C 180,E1 -14178.686,E2 -14178.686} C_VEL
LIN {X 0,Y 340.719,Z 295.667,A -85,B 0,C 180,E1 -14181.769,E2 -14181.769} C_VEL
LIN {X 0,Y 340.723,Z 295.655,A -85,B 0,C 180,E1 -14185.595,E2 -14185.595} C_VEL
LIN {X 0,Y 340.693,Z 295.67,A -85,B 0,C 180,E1 -14188.953,E2 -14188.953} C_VEL
LIN {X 0,Y 340.71,Z 295.664,A -85,B 0,C 180,E1 -14193.01,E2 -14193.01} C_VEL
LIN {X 0,Y 340.699,Z 295.669,A -85,B 0,C 180,E1 -14196.923,E2 -14196.923} C_VEL
LIN {X 0,Y 340.732,Z 295.663,A -85,B 0,C 180,E1 -14200.728,E2 -14200.728} C_VEL
LIN {X 0,Y 340.815,Z 295.652,A -85,B 0,C 180,E1 -14204.449,E2 -14204.449} C_VEL
LIN {X 0,Y 340.841,Z 295.625,A -85,B 0,C 180,E1 -14208.099,E2 -14208.099} C_VEL
LIN {X 0,Y 340.977,Z 295.638,A -85,B 0,C 180,E1 -14211.703,E2 -14211.703} C_VEL
LIN {X 0,Y 341.005,Z 295.624,A -85,B 0,C 180,E1 -14214.083,E2 -14214.083} C_VEL
LIN {X 0,Y 341.087,Z 295.595,A -85,B 0,C 180,E1 -14217.636,E2 -14217.636} C_VEL
LIN {X 0,Y 341.081,Z 295.622,A -85,B 0,C 180,E1 -14221.179,E2 -14221.179} C_VEL
LIN {X 0,Y 341.12,Z 295.615,A -85,B 0,C 180,E1 -14222.36,E2 -14222.36} C_VEL
LIN {X 0,Y 340.978,Z 295.602,A -85,B 0,C 180,E1 -14227.102,E2 -14227.102} C_VEL
LIN {X 0,Y 340.829,Z 295.651,A -85,B 0,C 180,E1 -14230.693,E2 -14230.693} C_VEL
LIN {X 0,Y 340.856,Z 295.64,A -85,B 0,C 180,E1 -14234.323,E2 -14234.323} C_VEL
LIN {X 0,Y 340.777,Z 295.64,A -85,B 0,C 180,E1 -14238.438,E2 -14238.438} C_VEL
LIN {X 0,Y 340.709,Z 295.669,A -85,B 0,C 180,E1 -14241.84,E2 -14241.84} C_VEL
LIN {X 0,Y 340.696,Z 295.659,A -85,B 0,C 180,E1 -14244.819,E2 -14244.819} C_VEL
LIN {X 0,Y 340.664,Z 295.653,A -85,B 0,C 180,E1 -14248.324,E2 -14248.324} C_VEL
LIN {X 0,Y 340.682,Z 295.671,A -85,B 0,C 180,E1 -14251.043,E2 -14251.043} C_VEL
LIN {X 0,Y 340.703,Z 295.65,A -85,B 0,C 180,E1 -14255.278,E2 -14255.278} C_VEL
LIN {X 0,Y 340.68,Z 295.658,A -85,B 0,C 180,E1 -14258.38,E2 -14258.38} C_VEL
LIN {X 0,Y 340.679,Z 295.672,A -85,B 0,C 180,E1 -14262.042,E2 -14262.042} C_VEL
LIN {X 0,Y 340.636,Z 295.661,A -85,B 0,C 180,E1 -14266.226,E2 -14266.226} C_VEL
LIN {X 0,Y 340.672,Z 295.675,A -85,B 0,C 180,E1 -14269.752,E2 -14269.752} C_VEL
LIN {X 0,Y 340.689,Z 295.656,A -85,B 0,C 180,E1 -14273.257,E2 -14273.257} C_VEL
LIN {X 0,Y 340.677,Z 295.674,A -85,B 0,C 180,E1 -14276.152,E2 -14276.152} C_VEL
LIN {X 0,Y 340.722,Z 295.654,A -85,B 0,C 180,E1 -14280.328,E2 -14280.328} C_VEL
LIN {X 0,Y 340.787,Z 295.659,A -85,B 0,C 180,E1 -14283.019,E2 -14283.019} C_VEL
LIN {X 0,Y 340.738,Z 295.659,A -85,B 0,C 180,E1 -14285.637,E2 -14285.637} C_VEL
LIN {X 0,Y 340.718,Z 295.66,A -85,B 0,C 180,E1 -14289.472,E2 -14289.472} C_VEL
LIN {X 0,Y 340.841,Z 295.655,A -85,B 0,C 180,E1 -14291.983,E2 -14291.983} C_VEL
LIN {X 0,Y 340.853,Z 295.651,A -85,B 0,C 180,E1 -14295.704,E2 -14295.704} C_VEL
LIN {X 0,Y 340.858,Z 295.646,A -85,B 0,C 180,E1 -14299.306,E2 -14299.306} C_VEL
LIN {X 0,Y 341.042,Z 295.629,A -85,B 0,C 180,E1 -14302.897,E2 -14302.897} C_VEL
LIN {X 0,Y 340.853,Z 295.791,A -85,B 0,C 180,E1 -14305.528,E2 -14305.528} C_VEL
LIN {X 0,Y 341.889,Z 299.281,A -85,B 0,C 180,E1 -14306.464,E2 -14306.464} C_VEL
LIN {X 0,Y 350.714,Z 316.973,A -85,B 0,C 180,E1 -14307.777,E2 -14307.777} C_VEL
LIN {X 0,Y 358.993,Z 336.389,A -85,B 0,C 180,E1 -14309.006,E2 -14309.006} C_VEL
LIN {X 0,Y 360.68,Z 341.097,A -85,B 0,C 180,E1 -14309.266,E2 -14309.266} C_VEL
LIN {X 0,Y 356.938,Z 463.922,A -85,B 0,C 180,E1 -14311.833,E2 -14311.833} C_VEL
LIN {X 0,Y 356.007,Z 480.048,A -85,B 0,C 180,E1 -14312.404,E2 -14312.404} C_VEL
LIN {X 0,Y 354.703,Z 495.488,A -85,B 0,C 180,E1 -14313.194,E2 -14313.194} C_VEL
LIN {X 0,Y 353.256,Z 509.405,A -85,B 0,C 180,E1 -14314.135,E2 -14314.135} C_VEL
LIN {X 0,Y 351.637,Z 522.638,A -85,B 0,C 180,E1 -14315.26,E2 -14315.26} C_VEL
LIN {X 0,Y 349.792,Z 535.759,A -85,B 0,C 180,E1 -14316.634,E2 -14316.634} C_VEL
LIN {X 0,Y 347.9,Z 547.947,A -85,B 0,C 180,E1 -14318.188,E2 -14318.188} C_VEL
LIN {X 0,Y 346.08,Z 559.3,A -85,B 0,C 180,E1 -14319.939,E2 -14319.939} C_VEL
LIN {X 0,Y 344.436,Z 569.197,A -85,B 0,C 180,E1 -14321.773,E2 -14321.773} C_VEL
LIN {X 0,Y 342.995,Z 577.608,A -85,B 0,C 180,E1 -14323.628,E2 -14323.628} C_VEL
LIN {X 0,Y 341.66,Z 585.847,A -85,B 0,C 180,E1 -14325.815,E2 -14325.815} C_VEL
LIN {X 0,Y 340.681,Z 592.624,A -85,B 0,C 180,E1 -14328.025,E2 -14328.025} C_VEL
LIN {X 0,Y 339.849,Z 598.812,A -85,B 0,C 180,E1 -14330.582,E2 -14330.582} C_VEL
LIN {X 0,Y 339.477,Z 602.47,A -85,B 0,C 180,E1 -14332.518,E2 -14332.518} C_VEL
LIN {X 0,Y 339.108,Z 605.25,A -85,B 0,C 180,E1 -14334.487,E2 -14334.487} C_VEL
LIN {X 0,Y 338.815,Z 607.753,A -85,B 0,C 180,E1 -14337.15,E2 -14337.15} C_VEL
LIN {X 0,Y 338.747,Z 608.468,A -85,B 0,C 180,E1 -14338.516,E2 -14338.516} C_VEL
LIN {X 0,Y 338.043,Z 608.783,A -85,B 0,C 180,E1 -14339.508,E2 -14339.508} C_VEL
LIN {X 0,Y 335.179,Z 608.892,A -85,B 0,C 180,E1 -14341.126,E2 -14341.126} C_VEL
LIN {X 0,Y 332.819,Z 608.635,A -85,B 0,C 180,E1 -14342.434,E2 -14342.434} C_VEL
LIN {X 0,Y 331.867,Z 608.2,A -85,B 0,C 180,E1 -14343.444,E2 -14343.444} C_VEL
LIN {X 0,Y 331.822,Z 607.978,A -85,B 0,C 180,E1 -14343.784,E2 -14343.784} C_VEL
LIN {X 0,Y 332.2,Z 605.509,A -85,B 0,C 180,E1 -14346.498,E2 -14346.498} C_VEL
LIN {X 0,Y 332.68,Z 602.605,A -85,B 0,C 180,E1 -14348.594,E2 -14348.594} C_VEL
LIN {X 0,Y 333.314,Z 598.466,A -85,B 0,C 180,E1 -14350.815,E2 -14350.815} C_VEL
LIN {X 0,Y 334.289,Z 592.813,A -85,B 0,C 180,E1 -14353.173,E2 -14353.173} C_VEL
LIN {X 0,Y 335.536,Z 586.11,A -85,B 0,C 180,E1 -14355.408,E2 -14355.408} C_VEL
LIN {X 0,Y 337.218,Z 577.591,A -85,B 0,C 180,E1 -14357.717,E2 -14357.717} C_VEL
LIN {X 0,Y 338.894,Z 568.973,A -85,B 0,C 180,E1 -14359.65,E2 -14359.65} C_VEL
LIN {X 0,Y 341.012,Z 558.768,A -85,B 0,C 180,E1 -14361.548,E2 -14361.548} C_VEL
LIN {X 0,Y 343.24,Z 547.114,A -85,B 0,C 180,E1 -14363.345,E2 -14363.345} C_VEL
LIN {X 0,Y 345.554,Z 534.245,A -85,B 0,C 180,E1 -14364.971,E2 -14364.971} C_VEL
LIN {X 0,Y 347.513,Z 521.934,A -85,B 0,C 180,E1 -14366.251,E2 -14366.251} C_VEL
LIN {X 0,Y 349.451,Z 508.239,A -85,B 0,C 180,E1 -14367.402,E2 -14367.402} C_VEL
LIN {X 0,Y 351.149,Z 493.611,A -85,B 0,C 180,E1 -14368.368,E2 -14368.368} C_VEL
LIN {X 0,Y 352.511,Z 478.489,A -85,B 0,C 180,E1 -14369.115,E2 -14369.115} C_VEL
LIN {X 0,Y 353.533,Z 463.56,A -85,B 0,C 180,E1 -14369.618,E2 -14369.618} C_VEL
LIN {X 0,Y 357.707,Z 344.537,A -85,B 0,C 180,E1 -14372.199,E2 -14372.199} C_VEL
LIN {X 0,Y 349.43,Z 326.643,A -85,B 0,C 180,E1 -14373.654,E2 -14373.654} C_VEL
LIN {X 0,Y 342.163,Z 313.09,A -85,B 0,C 180,E1 -14374.965,E2 -14374.965} C_VEL
LIN {X 0,Y 336.549,Z 303.803,A -85,B 0,C 180,E1 -14376.014,E2 -14376.014} C_VEL
LIN {X 0,Y 334.923,Z 300.822,A -85,B 0,C 180,E1 -14376.342,E2 -14376.342} C_VEL
LIN {X 0,Y 333.677,Z 296.543,A -85,B 0,C 180,E1 -14377.819,E2 -14377.819} C_VEL
LIN {X 0,Y 333.78,Z 296.53,A -85,B 0,C 180,E1 -14381.591,E2 -14381.591} C_VEL
LIN {X 0,Y 333.796,Z 296.531,A -85,B 0,C 180,E1 -14385.579,E2 -14385.579} C_VEL
LIN {X 0,Y 333.821,Z 296.526,A -85,B 0,C 180,E1 -14389.08,E2 -14389.08} C_VEL
LIN {X 0,Y 333.995,Z 296.508,A -85,B 0,C 180,E1 -14392.749,E2 -14392.749} C_VEL
LIN {X 0,Y 333.796,Z 296.533,A -85,B 0,C 180,E1 -14395.171,E2 -14395.171} C_VEL
LIN {X 0,Y 334.094,Z 296.495,A -85,B 0,C 180,E1 -14397.591,E2 -14397.591} C_VEL
LIN {X 0,Y 334.236,Z 296.475,A -85,B 0,C 180,E1 -14400.002,E2 -14400.002} C_VEL
LIN {X 0,Y 334.092,Z 296.489,A -85,B 0,C 180,E1 -14402.413,E2 -14402.413} C_VEL
LIN {X 0,Y 333.991,Z 296.506,A -85,B 0,C 180,E1 -14406.041,E2 -14406.041} C_VEL
LIN {X 0,Y 333.812,Z 296.529,A -85,B 0,C 180,E1 -14409.698,E2 -14409.698} C_VEL
LIN {X 0,Y 333.785,Z 296.528,A -85,B 0,C 180,E1 -14413.394,E2 -14413.394} C_VEL
LIN {X 0,Y 333.711,Z 296.536,A -85,B 0,C 180,E1 -14417.15,E2 -14417.15} C_VEL
LIN {X 0,Y 333.664,Z 296.544,A -85,B 0,C 180,E1 -14419.697,E2 -14419.697} C_VEL
LIN {X 0,Y 333.638,Z 296.546,A -85,B 0,C 180,E1 -14423.594,E2 -14423.594} C_VEL
LIN {X 0,Y 333.661,Z 296.547,A -85,B 0,C 180,E1 -14427.608,E2 -14427.608} C_VEL
LIN {X 0,Y 333.65,Z 296.549,A -85,B 0,C 180,E1 -14430.369,E2 -14430.369} C_VEL
LIN {X 0,Y 333.631,Z 296.549,A -85,B 0,C 180,E1 -14433.211,E2 -14433.211} C_VEL
LIN {X 0,Y 333.669,Z 296.544,A -85,B 0,C 180,E1 -14436.141,E2 -14436.141} C_VEL
LIN {X 0,Y 333.598,Z 296.549,A -85,B 0,C 180,E1 -14439.201,E2 -14439.201} C_VEL
LIN {X 0,Y 333.624,Z 296.554,A -85,B 0,C 180,E1 -14442.5,E2 -14442.5} C_VEL
LIN {X 0,Y 333.591,Z 296.555,A -85,B 0,C 180,E1 -14445.956,E2 -14445.956} C_VEL
LIN {X 0,Y 333.644,Z 296.558,A -85,B 0,C 180,E1 -14448.835,E2 -14448.835} C_VEL
LIN {X 0,Y 337.116,Z 307.908,A -85,B 0,C 180,E1 -14452.394,E2 -14452.394} C_VEL
LIN {X 0,Y 339.032,Z 314.579,A -85,B 0,C 180,E1 -14454.283,E2 -14454.283} C_VEL
LIN {X 0,Y 346.485,Z 329.022,A -85,B 0,C 180,E1 -14455.675,E2 -14455.675} C_VEL
LIN {X 0,Y 352.024,Z 340.753,A -85,B 0,C 180,E1 -14456.677,E2 -14456.677} C_VEL
LIN {X 0,Y 354.117,Z 345.736,A -85,B 0,C 180,E1 -14457.054,E2 -14457.054} C_VEL
LIN {X 0,Y 357.184,Z 364.034,A -85,B 0,C 180,E1 -14457.875,E2 -14457.875} C_VEL
LIN {X 0,Y 352.974,Z 482.14,A -85,B 0,C 180,E1 -14460.436,E2 -14460.436} C_VEL
LIN {X 0,Y 351.773,Z 497.631,A -85,B 0,C 180,E1 -14460.982,E2 -14460.982} C_VEL
LIN {X 0,Y 350.077,Z 513.206,A -85,B 0,C 180,E1 -14461.77,E2 -14461.77} C_VEL
LIN {X 0,Y 348.221,Z 527.721,A -85,B 0,C 180,E1 -14462.759,E2 -14462.759} C_VEL
LIN {X 0,Y 346.129,Z 541.556,A -85,B 0,C 180,E1 -14463.956,E2 -14463.956} C_VEL
LIN {X 0,Y 343.842,Z 554.914,A -85,B 0,C 180,E1 -14465.39,E2 -14465.39} C_VEL
LIN {X 0,Y 341.507,Z 567.12,A -85,B 0,C 180,E1 -14466.984,E2 -14466.984} C_VEL
LIN {X 0,Y 339.613,Z 577.542,A -85,B 0,C 180,E1 -14468.631,E2 -14468.631} C_VEL
LIN {X 0,Y 337.678,Z 587.716,A -85,B 0,C 180,E1 -14470.55,E2 -14470.55} C_VEL
LIN {X 0,Y 335.837,Z 597.009,A -85,B 0,C 180,E1 -14472.651,E2 -14472.651} C_VEL
LIN {X 0,Y 334.432,Z 604.767,A -85,B 0,C 180,E1 -14474.771,E2 -14474.771} C_VEL
LIN {X 0,Y 333.326,Z 612.032,A -85,B 0,C 180,E1 -14477.21,E2 -14477.21} C_VEL
LIN {X 0,Y 332.505,Z 617.783,A -85,B 0,C 180,E1 -14479.651,E2 -14479.651} C_VEL
LIN {X 0,Y 332.223,Z 621.237,A -85,B 0,C 180,E1 -14481.485,E2 -14481.485} C_VEL
LIN {X 0,Y 331.952,Z 625.114,A -85,B 0,C 180,E1 -14484.318,E2 -14484.318} C_VEL
LIN {X 0,Y 331.939,Z 626.857,A -85,B 0,C 180,E1 -14486.359,E2 -14486.359} C_VEL
LIN {X 0,Y 331.922,Z 627.895,A -85,B 0,C 180,E1 -14488.787,E2 -14488.787} C_VEL
LIN {X 0,Y 331.924,Z 627.779,A -85,B 0,C 180,E1 -14491.214,E2 -14491.214} C_VEL
LIN {X 0,Y 331.945,Z 626.481,A -85,B 0,C 180,E1 -14493.642,E2 -14493.642} C_VEL
LIN {X 0,Y 331.999,Z 623.944,A -85,B 0,C 180,E1 -14496.076,E2 -14496.076} C_VEL
LIN {X 0,Y 332.224,Z 620.164,A -85,B 0,C 180,E1 -14498.516,E2 -14498.516} C_VEL
LIN {X 0,Y 332.615,Z 615.039,A -85,B 0,C 180,E1 -14500.963,E2 -14500.963} C_VEL
LIN {X 0,Y 333.492,Z 608.447,A -85,B 0,C 180,E1 -14503.404,E2 -14503.404} C_VEL
LIN {X 0,Y 334.471,Z 601.322,A -85,B 0,C 180,E1 -14505.54,E2 -14505.54} C_VEL
LIN {X 0,Y 335.807,Z 592.74,A -85,B 0,C 180,E1 -14507.666,E2 -14507.666} C_VEL
LIN {X 0,Y 337.431,Z 584.045,A -85,B 0,C 180,E1 -14509.466,E2 -14509.466} C_VEL
LIN {X 0,Y 339.105,Z 573.48,A -85,B 0,C 180,E1 -14511.307,E2 -14511.307} C_VEL
LIN {X 0,Y 341.071,Z 561.428,A -85,B 0,C 180,E1 -14513.048,E2 -14513.048} C_VEL
LIN {X 0,Y 343.1,Z 549.103,A -85,B 0,C 180,E1 -14514.507,E2 -14514.507} C_VEL
LIN {X 0,Y 345.018,Z 535.684,A -85,B 0,C 180,E1 -14515.811,E2 -14515.811} C_VEL
LIN {X 0,Y 346.884,Z 521.086,A -85,B 0,C 180,E1 -14516.941,E2 -14516.941} C_VEL
LIN {X 0,Y 348.427,Z 506.605,A -85,B 0,C 180,E1 -14517.804,E2 -14517.804} C_VEL
LIN {X 0,Y 349.713,Z 491.331,A -85,B 0,C 180,E1 -14518.468,E2 -14518.468} C_VEL
LIN {X 0,Y 350.582,Z 475.357,A -85,B 0,C 180,E1 -14518.922,E2 -14518.922} C_VEL
LIN {X 0,Y 353.96,Z 363.064,A -85,B 0,C 180,E1 -14521.298,E2 -14521.298} C_VEL
LIN {X 0,Y 349.947,Z 341.074,A -85,B 0,C 180,E1 -14522.198,E2 -14522.198} C_VEL
LIN {X 0,Y 341.06,Z 320.894,A -85,B 0,C 180,E1 -14523.562,E2 -14523.562} C_VEL
LIN {X 0,Y 338.721,Z 315.656,A -85,B 0,C 180,E1 -14523.961,E2 -14523.961} C_VEL
LIN {X 0,Y 335.436,Z 302.897,A -85,B 0,C 180,E1 -14527.232,E2 -14527.232} C_VEL
LIN {X 0,Y 333.616,Z 296.558,A -85,B 0,C 180,E1 -14529.008,E2 -14529.008} C_VEL
LIN {X 0,Y 333.628,Z 296.549,A -85,B 0,C 180,E1 -14532.497,E2 -14532.497} C_VEL
LIN {X 0,Y 333.595,Z 296.552,A -85,B 0,C 180,E1 -14535.953,E2 -14535.953} C_VEL
LIN {X 0,Y 333.603,Z 296.559,A -85,B 0,C 180,E1 -14539.323,E2 -14539.323} C_VEL
LIN {X 0,Y 333.662,Z 296.552,A -85,B 0,C 180,E1 -14543.168,E2 -14543.168} C_VEL
LIN {X 0,Y 333.673,Z 296.534,A -85,B 0,C 180,E1 -14545.34,E2 -14545.34} C_VEL
LIN {X 0,Y 333.63,Z 296.552,A -85,B 0,C 180,E1 -14548.22,E2 -14548.22} C_VEL
LIN {X 0,Y 333.631,Z 296.551,A -85,B 0,C 180,E1 -14551.019,E2 -14551.019} C_VEL
LIN {X 0,Y 333.658,Z 296.55,A -85,B 0,C 180,E1 -14554.92,E2 -14554.92} C_VEL
LIN {X 0,Y 333.662,Z 296.551,A -85,B 0,C 180,E1 -14559.016,E2 -14559.016} C_VEL
LIN {X 0,Y 333.739,Z 296.539,A -85,B 0,C 180,E1 -14561.585,E2 -14561.585} C_VEL
LIN {X 0,Y 333.807,Z 296.511,A -85,B 0,C 180,E1 -14565.575,E2 -14565.575} C_VEL
LIN {X 0,Y 333.809,Z 296.51,A -85,B 0,C 180,E1 -14569.075,E2 -14569.075} C_VEL
LIN {X 0,Y 333.951,Z 296.51,A -85,B 0,C 180,E1 -14572.744,E2 -14572.744} C_VEL
LIN {X 0,Y 333.765,Z 296.516,A -85,B 0,C 180,E1 -14575.167,E2 -14575.167} C_VEL
LIN {X 0,Y 334.031,Z 296.472,A -85,B 0,C 180,E1 -14577.586,E2 -14577.586} C_VEL
LIN {X 0,Y 334.052,Z 296.498,A -85,B 0,C 180,E1 -14581.204,E2 -14581.204} C_VEL
LIN {X 0,Y 334.061,Z 296.495,A -85,B 0,C 180,E1 -14582.409,E2 -14582.409} C_VEL
LIN {X 0,Y 333.927,Z 296.478,A -85,B 0,C 180,E1 -14586.447,E2 -14586.447} C_VEL
LIN {X 0,Y 333.803,Z 296.523,A -85,B 0,C 180,E1 -14589.695,E2 -14589.695} C_VEL
LIN {X 0,Y 333.784,Z 296.527,A -85,B 0,C 180,E1 -14593.39,E2 -14593.39} C_VEL
LIN {X 0,Y 333.747,Z 296.507,A -85,B 0,C 180,E1 -14595.885,E2 -14595.885} C_VEL
LIN {X 0,Y 333.676,Z 296.535,A -85,B 0,C 180,E1 -14599.692,E2 -14599.692} C_VEL
LIN {X 0,Y 333.635,Z 296.545,A -85,B 0,C 180,E1 -14603.59,E2 -14603.59} C_VEL
LIN {X 0,Y 333.646,Z 296.518,A -85,B 0,C 180,E1 -14607.605,E2 -14607.605} C_VEL
LIN {X 0,Y 333.646,Z 296.543,A -85,B 0,C 180,E1 -14610.364,E2 -14610.364} C_VEL
LIN {X 0,Y 333.625,Z 296.55,A -85,B 0,C 180,E1 -14613.207,E2 -14613.207} C_VEL
LIN {X 0,Y 333.66,Z 296.521,A -85,B 0,C 180,E1 -14616.138,E2 -14616.138} C_VEL
LIN {X 0,Y 333.588,Z 296.548,A -85,B 0,C 180,E1 -14619.197,E2 -14619.197} C_VEL
LIN {X 0,Y 333.615,Z 296.553,A -85,B 0,C 180,E1 -14622.497,E2 -14622.497} C_VEL
LIN {X 0,Y 333.58,Z 296.537,A -85,B 0,C 180,E1 -14625.953,E2 -14625.953} C_VEL
LIN {X 0,Y 333.633,Z 296.554,A -85,B 0,C 180,E1 -14629.314,E2 -14629.314} C_VEL
LIN {X 0,Y 333.65,Z 296.532,A -85,B 0,C 180,E1 -14633.167,E2 -14633.167} C_VEL
LIN {X 0,Y 333.659,Z 296.549,A -85,B 0,C 180,E1 -14635.34,E2 -14635.34} C_VEL
LIN {X 0,Y 333.615,Z 296.548,A -85,B 0,C 180,E1 -14638.221,E2 -14638.221} C_VEL
LIN {X 0,Y 333.701,Z 296.542,A -85,B 0,C 180,E1 -14642.19,E2 -14642.19} C_VEL
LIN {X 0,Y 333.709,Z 296.531,A -85,B 0,C 180,E1 -14645.089,E2 -14645.089} C_VEL
LIN {X 0,Y 333.657,Z 296.541,A -85,B 0,C 180,E1 -14649.018,E2 -14649.018} C_VEL
LIN {X 0,Y 333.777,Z 296.535,A -85,B 0,C 180,E1 -14651.588,E2 -14651.588} C_VEL
LIN {X 0,Y 333.792,Z 296.53,A -85,B 0,C 180,E1 -14655.576,E2 -14655.576} C_VEL
LIN {X 0,Y 333.821,Z 296.524,A -85,B 0,C 180,E1 -14659.077,E2 -14659.077} C_VEL
LIN {X 0,Y 333.995,Z 296.506,A -85,B 0,C 180,E1 -14662.747,E2 -14662.747} C_VEL
LIN {X 0,Y 333.835,Z 296.647,A -85,B 0,C 180,E1 -14664.942,E2 -14664.942} C_VEL
LIN {X 0,Y 334.589,Z 299.565,A -85,B 0,C 180,E1 -14665.713,E2 -14665.713} C_VEL
LIN {X 0,Y 341.868,Z 313.716,A -85,B 0,C 180,E1 -14666.83,E2 -14666.83} C_VEL
LIN {X 0,Y 348.117,Z 327.219,A -85,B 0,C 180,E1 -14667.78,E2 -14667.78} C_VEL
LIN {X 0,Y 354.311,Z 342.245,A -85,B 0,C 180,E1 -14668.725,E2 -14668.725} C_VEL
LIN {X 0,Y 351.65,Z 430.369,A -85,B 0,C 180,E1 -14670.587,E2 -14670.587} C_VEL
LIN {X 0,Y 350.538,Z 465.253,A -85,B 0,C 180,E1 -14671.364,E2 -14671.364} C_VEL
LIN {X 0,Y 349.599,Z 480.273,A -85,B 0,C 180,E1 -14671.908,E2 -14671.908} C_VEL
LIN {X 0,Y 348.319,Z 495.115,A -85,B 0,C 180,E1 -14672.674,E2 -14672.674} C_VEL
LIN {X 0,Y 346.874,Z 508.923,A -85,B 0,C 180,E1 -14673.615,E2 -14673.615} C_VEL
LIN {X 0,Y 345.074,Z 522.922,A -85,B 0,C 180,E1 -14674.819,E2 -14674.819} C_VEL
LIN {X 0,Y 343.005,Z 536.915,A -85,B 0,C 180,E1 -14676.322,E2 -14676.322} C_VEL
LIN {X 0,Y 340.985,Z 549.587,A -85,B 0,C 180,E1 -14678.002,E2 -14678.002} C_VEL
LIN {X 0,Y 339.06,Z 561.039,A -85,B 0,C 180,E1 -14679.846,E2 -14679.846} C_VEL
LIN {X 0,Y 337.348,Z 570.821,A -85,B 0,C 180,E1 -14681.734,E2 -14681.734} C_VEL
LIN {X 0,Y 335.716,Z 580.206,A -85,B 0,C 180,E1 -14683.93,E2 -14683.93} C_VEL
LIN {X 0,Y 334.409,Z 588.05,A -85,B 0,C 180,E1 -14686.168,E2 -14686.168} C_VEL
LIN {X 0,Y 333.43,Z 594.595,A -85,B 0,C 180,E1 -14688.477,E2 -14688.477} C_VEL
LIN {X 0,Y 332.673,Z 600.288,A -85,B 0,C 180,E1 -14691.046,E2 -14691.046} C_VEL
LIN {X 0,Y 332.41,Z 602.621,A -85,B 0,C 180,E1 -14692.368,E2 -14692.368} C_VEL
LIN {X 0,Y 331.924,Z 606.216,A -85,B 0,C 180,E1 -14695.053,E2 -14695.053} C_VEL
LIN {X 0,Y 331.676,Z 608.371,A -85,B 0,C 180,E1 -14697.784,E2 -14697.784} C_VEL
LIN {X 0,Y 331.645,Z 608.978,A -85,B 0,C 180,E1 -14699.681,E2 -14699.681} C_VEL
LIN {X 0,Y 331.701,Z 608.806,A -85,B 0,C 180,E1 -14702.064,E2 -14702.064} C_VEL
LIN {X 0,Y 331.822,Z 607.978,A -85,B 0,C 180,E1 -14703.784,E2 -14703.784} C_VEL
LIN {X 0,Y 331.283,Z 607.295,A -85,B 0,C 180,E1 -14704.793,E2 -14704.793} C_VEL
LIN {X 0,Y 328.678,Z 605.857,A -85,B 0,C 180,E1 -14706.436,E2 -14706.436} C_VEL
LIN {X 0,Y 326.51,Z 604.344,A -85,B 0,C 180,E1 -14707.754,E2 -14707.754} C_VEL
LIN {X 0,Y 325.693,Z 602.917,A -85,B 0,C 180,E1 -14708.758,E2 -14708.758} C_VEL
LIN {X 0,Y 325.689,Z 602.358,A -85,B 0,C 180,E1 -14709.093,E2 -14709.093} C_VEL
LIN {X 0,Y 326.611,Z 597.053,A -85,B 0,C 180,E1 -14711.838,E2 -14711.838} C_VEL
LIN {X 0,Y 327.712,Z 591.177,A -85,B 0,C 180,E1 -14714.184,E2 -14714.184} C_VEL
LIN {X 0,Y 329.186,Z 583.81,A -85,B 0,C 180,E1 -14716.541,E2 -14716.541} C_VEL
LIN {X 0,Y 331.1,Z 574.857,A -85,B 0,C 180,E1 -14718.855,E2 -14718.855} C_VEL
LIN {X 0,Y 333.163,Z 565.184,A -85,B 0,C 180,E1 -14720.91,E2 -14720.91} C_VEL
LIN {X 0,Y 335.402,Z 554.599,A -85,B 0,C 180,E1 -14722.771,E2 -14722.771} C_VEL
LIN {X 0,Y 337.697,Z 542.846,A -85,B 0,C 180,E1 -14724.485,E2 -14724.485} C_VEL
LIN {X 0,Y 339.925,Z 530.597,A -85,B 0,C 180,E1 -14725.961,E2 -14725.961} C_VEL
LIN {X 0,Y 341.913,Z 518.283,A -85,B 0,C 180,E1 -14727.178,E2 -14727.178} C_VEL
LIN {X 0,Y 343.956,Z 503.807,A -85,B 0,C 180,E1 -14728.33,E2 -14728.33} C_VEL
LIN {X 0,Y 345.567,Z 489.395,A -85,B 0,C 180,E1 -14729.218,E2 -14729.218} C_VEL
LIN {X 0,Y 346.861,Z 474.526,A -85,B 0,C 180,E1 -14729.892,E2 -14729.892} C_VEL
LIN {X 0,Y 347.748,Z 459.616,A -85,B 0,C 180,E1 -14730.343,E2 -14730.343} C_VEL
LIN {X 0,Y 351.905,Z 346.731,A -85,B 0,C 180,E1 -14732.813,E2 -14732.813} C_VEL
LIN {X 0,Y 343.28,Z 328.22,A -85,B 0,C 180,E1 -14734.392,E2 -14734.392} C_VEL
LIN {X 0,Y 335.236,Z 313.575,A -85,B 0,C 180,E1 -14735.914,E2 -14735.914} C_VEL
LIN {X 0,Y 329.322,Z 304.038,A -85,B 0,C 180,E1 -14737.081,E2 -14737.081} C_VEL
LIN {X 0,Y 327.706,Z 301.049,A -85,B 0,C 180,E1 -14737.45,E2 -14737.45} C_VEL
LIN {X 0,Y 326.631,Z 297.426,A -85,B 0,C 180,E1 -14738.795,E2 -14738.795} C_VEL
LIN {X 0,Y 326.732,Z 297.405,A -85,B 0,C 180,E1 -14741.179,E2 -14741.179} C_VEL
LIN {X 0,Y 326.751,Z 297.408,A -85,B 0,C 180,E1 -14745.435,E2 -14745.435} C_VEL
LIN {X 0,Y 326.757,Z 297.407,A -85,B 0,C 180,E1 -14748.841,E2 -14748.841} C_VEL
LIN {X 0,Y 326.947,Z 297.385,A -85,B 0,C 180,E1 -14752.592,E2 -14752.592} C_VEL
LIN {X 0,Y 326.763,Z 297.409,A -85,B 0,C 180,E1 -14755.067,E2 -14755.067} C_VEL
LIN {X 0,Y 327.034,Z 297.374,A -85,B 0,C 180,E1 -14757.539,E2 -14757.539} C_VEL
LIN {X 0,Y 327.188,Z 297.353,A -85,B 0,C 180,E1 -14760.002,E2 -14760.002} C_VEL
LIN {X 0,Y 327.033,Z 297.368,A -85,B 0,C 180,E1 -14762.465,E2 -14762.465} C_VEL
LIN {X 0,Y 326.945,Z 297.384,A -85,B 0,C 180,E1 -14766.172,E2 -14766.172} C_VEL
LIN {X 0,Y 326.775,Z 297.405,A -85,B 0,C 180,E1 -14769.909,E2 -14769.909} C_VEL
LIN {X 0,Y 326.749,Z 297.404,A -85,B 0,C 180,E1 -14773.688,E2 -14773.688} C_VEL
LIN {X 0,Y 326.657,Z 297.415,A -85,B 0,C 180,E1 -14777.532,E2 -14777.532} C_VEL
LIN {X 0,Y 326.608,Z 297.426,A -85,B 0,C 180,E1 -14781.459,E2 -14781.459} C_VEL
LIN {X 0,Y 326.597,Z 297.424,A -85,B 0,C 180,E1 -14785.493,E2 -14785.493} C_VEL
LIN {X 0,Y 326.588,Z 297.425,A -85,B 0,C 180,E1 -14788.259,E2 -14788.259} C_VEL
LIN {X 0,Y 326.562,Z 297.426,A -85,B 0,C 180,E1 -14791.1,E2 -14791.1} C_VEL
LIN {X 0,Y 326.602,Z 297.422,A -85,B 0,C 180,E1 -14794.022,E2 -14794.022} C_VEL
LIN {X 0,Y 326.618,Z 297.42,A -85,B 0,C 180,E1 -14797.239,E2 -14797.239} C_VEL
LIN {X 0,Y 326.54,Z 297.431,A -85,B 0,C 180,E1 -14801.126,E2 -14801.126} C_VEL
LIN {X 0,Y 326.556,Z 297.43,A -85,B 0,C 180,E1 -14803.528,E2 -14803.528} C_VEL
LIN {X 0,Y 326.592,Z 297.463,A -85,B 0,C 180,E1 -14807.881,E2 -14807.881} C_VEL
LIN {X 0,Y 330.015,Z 308.47,A -85,B 0,C 180,E1 -14811.508,E2 -14811.508} C_VEL
LIN {X 0,Y 331.755,Z 314.294,A -85,B 0,C 180,E1 -14813.234,E2 -14813.234} C_VEL
LIN {X 0,Y 339.345,Z 328.528,A -85,B 0,C 180,E1 -14814.727,E2 -14814.727} C_VEL
LIN {X 0,Y 346.941,Z 344.545,A -85,B 0,C 180,E1 -14816.156,E2 -14816.156} C_VEL
LIN {X 0,Y 348.62,Z 348.727,A -85,B 0,C 180,E1 -14816.477,E2 -14816.477} C_VEL
LIN {X 0,Y 351.35,Z 365.123,A -85,B 0,C 180,E1 -14817.24,E2 -14817.24} C_VEL
LIN {X 0,Y 347.031,Z 481.319,A -85,B 0,C 180,E1 -14819.794,E2 -14819.794} C_VEL
LIN {X 0,Y 345.782,Z 497.012,A -85,B 0,C 180,E1 -14820.346,E2 -14820.346} C_VEL
LIN {X 0,Y 343.99,Z 512.662,A -85,B 0,C 180,E1 -14821.141,E2 -14821.141} C_VEL
LIN {X 0,Y 342.082,Z 527.154,A -85,B 0,C 180,E1 -14822.139,E2 -14822.139} C_VEL
LIN {X 0,Y 339.992,Z 540.348,A -85,B 0,C 180,E1 -14823.283,E2 -14823.283} C_VEL
LIN {X 0,Y 337.629,Z 553.868,A -85,B 0,C 180,E1 -14824.741,E2 -14824.741} C_VEL
LIN {X 0,Y 335.176,Z 566.209,A -85,B 0,C 180,E1 -14826.359,E2 -14826.359} C_VEL
LIN {X 0,Y 332.816,Z 578.278,A -85,B 0,C 180,E1 -14828.304,E2 -14828.304} C_VEL
LIN {X 0,Y 330.961,Z 587.732,A -85,B 0,C 180,E1 -14830.139,E2 -14830.139} C_VEL
LIN {X 0,Y 329.245,Z 595.741,A -85,B 0,C 180,E1 -14831.971,E2 -14831.971} C_VEL
LIN {X 0,Y 327.675,Z 603.677,A -85,B 0,C 180,E1 -14834.13,E2 -14834.13} C_VEL
LIN {X 0,Y 326.569,Z 610.288,A -85,B 0,C 180,E1 -14836.307,E2 -14836.307} C_VEL
LIN {X 0,Y 325.62,Z 616.386,A -85,B 0,C 180,E1 -14838.8,E2 -14838.8} C_VEL
LIN {X 0,Y 325.142,Z 621.098,A -85,B 0,C 180,E1 -14841.298,E2 -14841.298} C_VEL
LIN {X 0,Y 324.874,Z 624.495,A -85,B 0,C 180,E1 -14843.791,E2 -14843.791} C_VEL
LIN {X 0,Y 324.844,Z 626.679,A -85,B 0,C 180,E1 -14846.279,E2 -14846.279} C_VEL
LIN {X 0,Y 324.831,Z 627.696,A -85,B 0,C 180,E1 -14848.761,E2 -14848.761} C_VEL
LIN {X 0,Y 324.832,Z 627.558,A -85,B 0,C 180,E1 -14851.24,E2 -14851.24} C_VEL
LIN {X 0,Y 324.852,Z 626.245,A -85,B 0,C 180,E1 -14853.722,E2 -14853.722} C_VEL
LIN {X 0,Y 324.902,Z 623.686,A -85,B 0,C 180,E1 -14856.209,E2 -14856.209} C_VEL
LIN {X 0,Y 325.141,Z 619.878,A -85,B 0,C 180,E1 -14858.703,E2 -14858.703} C_VEL
LIN {X 0,Y 325.59,Z 614.725,A -85,B 0,C 180,E1 -14861.202,E2 -14861.202} C_VEL
LIN {X 0,Y 326.519,Z 608.1,A -85,B 0,C 180,E1 -14863.696,E2 -14863.696} C_VEL
LIN {X 0,Y 327.566,Z 600.94,A -85,B 0,C 180,E1 -14865.876,E2 -14865.876} C_VEL
LIN {X 0,Y 328.95,Z 592.316,A -85,B 0,C 180,E1 -14868.047,E2 -14868.047} C_VEL
LIN {X 0,Y 330.967,Z 581.935,A -85,B 0,C 180,E1 -14870.186,E2 -14870.186} C_VEL
LIN {X 0,Y 332.493,Z 572.563,A -85,B 0,C 180,E1 -14871.824,E2 -14871.824} C_VEL
LIN {X 0,Y 334.463,Z 560.862,A -85,B 0,C 180,E1 -14873.531,E2 -14873.531} C_VEL
LIN {X 0,Y 336.578,Z 548.47,A -85,B 0,C 180,E1 -14875.014,E2 -14875.014} C_VEL
LIN {X 0,Y 338.601,Z 534.958,A -85,B 0,C 180,E1 -14876.338,E2 -14876.338} C_VEL
LIN {X 0,Y 340.534,Z 519.953,A -85,B 0,C 180,E1 -14877.506,E2 -14877.506} C_VEL
LIN {X 0,Y 342.106,Z 505.543,A -85,B 0,C 180,E1 -14878.363,E2 -14878.363} C_VEL
LIN {X 0,Y 343.465,Z 489.91,A -85,B 0,C 180,E1 -14879.034,E2 -14879.034} C_VEL
LIN {X 0,Y 344.258,Z 474.69,A -85,B 0,C 180,E1 -14879.463,E2 -14879.463} C_VEL
LIN {X 0,Y 347.74,Z 364.208,A -85,B 0,C 180,E1 -14881.837,E2 -14881.837} C_VEL
LIN {X 0,Y 344.137,Z 343.963,A -85,B 0,C 180,E1 -14882.679,E2 -14882.679} C_VEL
LIN {X 0,Y 335.6,Z 324.476,A -85,B 0,C 180,E1 -14884.027,E2 -14884.027} C_VEL
LIN {X 0,Y 331.423,Z 315.396,A -85,B 0,C 180,E1 -14884.744,E2 -14884.744} C_VEL
LIN {X 0,Y 328.239,Z 303.242,A -85,B 0,C 180,E1 -14887.962,E2 -14887.962} C_VEL
LIN {X 0,Y 326.56,Z 297.434,A -85,B 0,C 180,E1 -14889.596,E2 -14889.596} C_VEL
LIN {X 0,Y 326.56,Z 297.425,A -85,B 0,C 180,E1 -14893.525,E2 -14893.525} C_VEL
LIN {X 0,Y 326.573,Z 297.426,A -85,B 0,C 180,E1 -14897.028,E2 -14897.028} C_VEL
LIN {X 0,Y 326.572,Z 297.423,A -85,B 0,C 180,E1 -14900.78,E2 -14900.78} C_VEL
LIN {X 0,Y 326.611,Z 297.42,A -85,B 0,C 180,E1 -14904.478,E2 -14904.478} C_VEL
LIN {X 0,Y 326.609,Z 297.423,A -85,B 0,C 180,E1 -14907.454,E2 -14907.454} C_VEL
LIN {X 0,Y 326.581,Z 297.43,A -85,B 0,C 180,E1 -14910.331,E2 -14910.331} C_VEL
LIN {X 0,Y 326.597,Z 297.423,A -85,B 0,C 180,E1 -14913.133,E2 -14913.133} C_VEL
LIN {X 0,Y 326.59,Z 297.428,A -85,B 0,C 180,E1 -14917.209,E2 -14917.209} C_VEL
LIN {X 0,Y 326.671,Z 297.416,A -85,B 0,C 180,E1 -14921.192,E2 -14921.192} C_VEL
LIN {X 0,Y 326.761,Z 297.39,A -85,B 0,C 180,E1 -14925.432,E2 -14925.432} C_VEL
LIN {X 0,Y 326.75,Z 297.388,A -85,B 0,C 180,E1 -14928.836,E2 -14928.836} C_VEL
LIN {X 0,Y 326.908,Z 297.387,A -85,B 0,C 180,E1 -14932.587,E2 -14932.587} C_VEL
LIN {X 0,Y 326.734,Z 297.392,A -85,B 0,C 180,E1 -14935.062,E2 -14935.062} C_VEL
LIN {X 0,Y 327.035,Z 297.358,A -85,B 0,C 180,E1 -14938.767,E2 -14938.767} C_VEL
LIN {X 0,Y 327.004,Z 297.374,A -85,B 0,C 180,E1 -14942.461,E2 -14942.461} C_VEL
LIN {X 0,Y 326.89,Z 297.354,A -85,B 0,C 180,E1 -14946.437,E2 -14946.437} C_VEL
LIN {X 0,Y 326.768,Z 297.402,A -85,B 0,C 180,E1 -14949.905,E2 -14949.905} C_VEL
LIN {X 0,Y 326.749,Z 297.4,A -85,B 0,C 180,E1 -14953.683,E2 -14953.683} C_VEL
LIN {X 0,Y 326.653,Z 297.387,A -85,B 0,C 180,E1 -14957.528,E2 -14957.528} C_VEL
LIN {X 0,Y 326.619,Z 297.418,A -85,B 0,C 180,E1 -14960.135,E2 -14960.135} C_VEL
LIN {X 0,Y 326.601,Z 297.418,A -85,B 0,C 180,E1 -14964.13,E2 -14964.13} C_VEL
LIN {X 0,Y 326.579,Z 297.404,A -85,B 0,C 180,E1 -14968.255,E2 -14968.255} C_VEL
LIN {X 0,Y 326.562,Z 297.43,A -85,B 0,C 180,E1 -14971.095,E2 -14971.095} C_VEL
LIN {X 0,Y 326.594,Z 297.42,A -85,B 0,C 180,E1 -14974.018,E2 -14974.018} C_VEL
LIN {X 0,Y 326.609,Z 297.398,A -85,B 0,C 180,E1 -14977.235,E2 -14977.235} C_VEL
LIN {X 0,Y 326.531,Z 297.44,A -85,B 0,C 180,E1 -14981.123,E2 -14981.123} C_VEL
LIN {X 0,Y 326.546,Z 297.423,A -85,B 0,C 180,E1 -14983.524,E2 -14983.524} C_VEL
LIN {X 0,Y 326.561,Z 297.42,A -85,B 0,C 180,E1 -14987.027,E2 -14987.027} C_VEL
LIN {X 0,Y 326.597,Z 297.426,A -85,B 0,C 180,E1 -14990.771,E2 -14990.771} C_VEL
LIN {X 0,Y 326.597,Z 297.418,A -85,B 0,C 180,E1 -14994.479,E2 -14994.479} C_VEL
LIN {X 0,Y 326.593,Z 297.426,A -85,B 0,C 180,E1 -14997.454,E2 -14997.454} C_VEL
LIN {X 0,Y 326.617,Z 297.411,A -85,B 0,C 180,E1 -15000.337,E2 -15000.337} C_VEL
LIN {X 0,Y 326.667,Z 297.417,A -85,B 0,C 180,E1 -15003.141,E2 -15003.141} C_VEL
LIN {X 0,Y 326.633,Z 297.417,A -85,B 0,C 180,E1 -15005.87,E2 -15005.87} C_VEL
LIN {X 0,Y 326.641,Z 297.413,A -85,B 0,C 180,E1 -15009.864,E2 -15009.864} C_VEL
LIN {X 0,Y 326.683,Z 297.416,A -85,B 0,C 180,E1 -15012.471,E2 -15012.471} C_VEL
LIN {X 0,Y 326.744,Z 297.405,A -85,B 0,C 180,E1 -15016.314,E2 -15016.314} C_VEL
LIN {X 0,Y 326.798,Z 297.399,A -85,B 0,C 180,E1 -15020.093,E2 -15020.093} C_VEL
LIN {X 0,Y 326.949,Z 297.382,A -85,B 0,C 180,E1 -15022.589,E2 -15022.589} C_VEL
LIN {X 0,Y 326.899,Z 297.475,A -85,B 0,C 180,E1 -15024.332,E2 -15024.332} C_VEL
LIN {X 0,Y 327.314,Z 299.586,A -85,B 0,C 180,E1 -15024.918,E2 -15024.918} C_VEL
LIN {X 0,Y 336.811,Z 318.154,A -85,B 0,C 180,E1 -15026.43,E2 -15026.43} C_VEL
LIN {X 0,Y 344.731,Z 335.635,A -85,B 0,C 180,E1 -15027.663,E2 -15027.663} C_VEL
LIN {X 0,Y 348.177,Z 344.503,A -85,B 0,C 180,E1 -15028.211,E2 -15028.211} C_VEL
LIN {X 0,Y 344.24,Z 464.472,A -85,B 0,C 180,E1 -15030.807,E2 -15030.807} C_VEL
LIN {X 0,Y 343.235,Z 480.47,A -85,B 0,C 180,E1 -15031.393,E2 -15031.393} C_VEL
LIN {X 0,Y 341.846,Z 495.895,A -85,B 0,C 180,E1 -15032.209,E2 -15032.209} C_VEL
LIN {X 0,Y 340.441,Z 508.83,A -85,B 0,C 180,E1 -15033.106,E2 -15033.106} C_VEL
LIN {X 0,Y 338.619,Z 522.594,A -85,B 0,C 180,E1 -15034.302,E2 -15034.302} C_VEL
LIN {X 0,Y 336.683,Z 535.5,A -85,B 0,C 180,E1 -15035.69,E2 -15035.69} C_VEL
LIN {X 0,Y 334.733,Z 547.339,A -85,B 0,C 180,E1 -15037.236,E2 -15037.236} C_VEL
LIN {X 0,Y 332.941,Z 557.406,A -85,B 0,C 180,E1 -15038.802,E2 -15038.802} C_VEL
LIN {X 0,Y 331.108,Z 567.678,A -85,B 0,C 180,E1 -15040.703,E2 -15040.703} C_VEL
LIN {X 0,Y 329.272,Z 577.708,A -85,B 0,C 180,E1 -15042.95,E2 -15042.95} C_VEL
LIN {X 0,Y 327.8,Z 586.117,A -85,B 0,C 180,E1 -15045.26,E2 -15045.26} C_VEL
LIN {X 0,Y 326.705,Z 592.839,A -85,B 0,C 180,E1 -15047.527,E2 -15047.527} C_VEL
LIN {X 0,Y 325.972,Z 597.699,A -85,B 0,C 180,E1 -15049.522,E2 -15049.522} C_VEL
LIN {X 0,Y 325.446,Z 602.043,A -85,B 0,C 180,E1 -15051.793,E2 -15051.793} C_VEL
LIN {X 0,Y 324.896,Z 606.096,A -85,B 0,C 180,E1 -15054.705,E2 -15054.705} C_VEL
LIN {X 0,Y 324.599,Z 608.364,A -85,B 0,C 180,E1 -15057.42,E2 -15057.42} C_VEL
LIN {X 0,Y 324.548,Z 609.221,A -85,B 0,C 180,E1 -15059.987,E2 -15059.987} C_VEL
LIN {X 0,Y 324.651,Z 608.786,A -85,B 0,C 180,E1 -15062.764,E2 -15062.764} C_VEL
LIN {X 0,Y 324.844,Z 607.655,A -85,B 0,C 180,E1 -15064.707,E2 -15064.707} C_VEL
LIN {X 0,Y 325.238,Z 605.088,A -85,B 0,C 180,E1 -15067.231,E2 -15067.231} C_VEL
LIN {X 0,Y 325.689,Z 602.358,A -85,B 0,C 180,E1 -15069.093,E2 -15069.093} C_VEL
LIN {X 0,Y 325.297,Z 600.722,A -85,B 0,C 180,E1 -15070.088,E2 -15070.088} C_VEL
LIN {X 0,Y 323.016,Z 597.779,A -85,B 0,C 180,E1 -15071.716,E2 -15071.716} C_VEL
LIN {X 0,Y 321.174,Z 595.168,A -85,B 0,C 180,E1 -15073.012,E2 -15073.012} C_VEL
LIN {X 0,Y 320.626,Z 592.882,A -85,B 0,C 180,E1 -15073.984,E2 -15073.984} C_VEL
LIN {X 0,Y 320.714,Z 592.042,A -85,B 0,C 180,E1 -15074.304,E2 -15074.304} C_VEL
LIN {X 0,Y 322.334,Z 584.4,A -85,B 0,C 180,E1 -15076.841,E2 -15076.841} C_VEL
LIN {X 0,Y 324.417,Z 575.083,A -85,B 0,C 180,E1 -15079.305,E2 -15079.305} C_VEL
LIN {X 0,Y 326.578,Z 565.471,A -85,B 0,C 180,E1 -15081.389,E2 -15081.389} C_VEL
LIN {X 0,Y 328.884,Z 555.112,A -85,B 0,C 180,E1 -15083.252,E2 -15083.252} C_VEL
LIN {X 0,Y 331.394,Z 542.854,A -85,B 0,C 180,E1 -15085.072,E2 -15085.072} C_VEL
LIN {X 0,Y 333.689,Z 530.828,A -85,B 0,C 180,E1 -15086.541,E2 -15086.541} C_VEL
LIN {X 0,Y 335.98,Z 517.157,A -85,B 0,C 180,E1 -15087.903,E2 -15087.903} C_VEL
LIN {X 0,Y 338.055,Z 502.704,A -85,B 0,C 180,E1 -15089.041,E2 -15089.041} C_VEL
LIN {X 0,Y 339.63,Z 488.638,A -85,B 0,C 180,E1 -15089.906,E2 -15089.906} C_VEL
LIN {X 0,Y 341.041,Z 473.061,A -85,B 0,C 180,E1 -15090.596,E2 -15090.596} C_VEL
LIN {X 0,Y 341.903,Z 457.205,A -85,B 0,C 180,E1 -15091.056,E2 -15091.056} C_VEL
LIN {X 0,Y 346.08,Z 348.905,A -85,B 0,C 180,E1 -15093.466,E2 -15093.466} C_VEL
LIN {X 0,Y 338.668,Z 332.837,A -85,B 0,C 180,E1 -15094.875,E2 -15094.875} C_VEL
LIN {X 0,Y 330.862,Z 318.381,A -85,B 0,C 180,E1 -15096.408,E2 -15096.408} C_VEL
LIN {X 0,Y 322.734,Z 305.106,A -85,B 0,C 180,E1 -15098.095,E2 -15098.095} C_VEL
LIN {X 0,Y 320.494,Z 301.367,A -85,B 0,C 180,E1 -15098.622,E2 -15098.622} C_VEL
LIN {X 0,Y 319.615,Z 298.298,A -85,B 0,C 180,E1 -15099.824,E2 -15099.824} C_VEL
LIN {X 0,Y 319.66,Z 298.293,A -85,B 0,C 180,E1 -15103.395,E2 -15103.395} C_VEL
LIN {X 0,Y 319.72,Z 298.286,A -85,B 0,C 180,E1 -15106.01,E2 -15106.01} C_VEL
LIN {X 0,Y 319.741,Z 298.282,A -85,B 0,C 180,E1 -15109.875,E2 -15109.875} C_VEL
LIN {X 0,Y 319.901,Z 298.262,A -85,B 0,C 180,E1 -15112.428,E2 -15112.428} C_VEL
LIN {X 0,Y 319.733,Z 298.283,A -85,B 0,C 180,E1 -15114.958,E2 -15114.958} C_VEL
LIN {X 0,Y 319.978,Z 298.254,A -85,B 0,C 180,E1 -15117.484,E2 -15117.484} C_VEL
LIN {X 0,Y 320.14,Z 298.231,A -85,B 0,C 180,E1 -15120.002,E2 -15120.002} C_VEL
LIN {X 0,Y 319.976,Z 298.247,A -85,B 0,C 180,E1 -15122.52,E2 -15122.52} C_VEL
LIN {X 0,Y 319.902,Z 298.262,A -85,B 0,C 180,E1 -15126.308,E2 -15126.308} C_VEL
LIN {X 0,Y 319.727,Z 298.283,A -85,B 0,C 180,E1 -15130.13,E2 -15130.13} C_VEL
LIN {X 0,Y 319.723,Z 298.278,A -85,B 0,C 180,E1 -15133.994,E2 -15133.994} C_VEL
LIN {X 0,Y 319.607,Z 298.295,A -85,B 0,C 180,E1 -15137.932,E2 -15137.932} C_VEL
LIN {X 0,Y 319.559,Z 298.306,A -85,B 0,C 180,E1 -15141.957,E2 -15141.957} C_VEL
LIN {X 0,Y 319.547,Z 298.3,A -85,B 0,C 180,E1 -15146.098,E2 -15146.098} C_VEL
LIN {X 0,Y 319.521,Z 298.302,A -85,B 0,C 180,E1 -15148.942,E2 -15148.942} C_VEL
LIN {X 0,Y 319.515,Z 298.302,A -85,B 0,C 180,E1 -15151.865,E2 -15151.865} C_VEL
LIN {X 0,Y 319.574,Z 298.301,A -85,B 0,C 180,E1 -15155.544,E2 -15155.544} C_VEL
LIN {X 0,Y 319.526,Z 298.304,A -85,B 0,C 180,E1 -15159.664,E2 -15159.664} C_VEL
LIN {X 0,Y 319.516,Z 298.307,A -85,B 0,C 180,E1 -15163.462,E2 -15163.462} C_VEL
LIN {X 0,Y 319.571,Z 298.483,A -85,B 0,C 180,E1 -15166.903,E2 -15166.903} C_VEL
LIN {X 0,Y 322.528,Z 307.726,A -85,B 0,C 180,E1 -15170.128,E2 -15170.128} C_VEL
LIN {X 0,Y 324.382,Z 313.864,A -85,B 0,C 180,E1 -15172.085,E2 -15172.085} C_VEL
LIN {X 0,Y 326.954,Z 318.416,A -85,B 0,C 180,E1 -15172.631,E2 -15172.631} C_VEL
LIN {X 0,Y 334.526,Z 332.616,A -85,B 0,C 180,E1 -15174.178,E2 -15174.178} C_VEL
LIN {X 0,Y 341.858,Z 348.273,A -85,B 0,C 180,E1 -15175.615,E2 -15175.615} C_VEL
LIN {X 0,Y 343.273,Z 352.148,A -85,B 0,C 180,E1 -15175.903,E2 -15175.903} C_VEL
LIN {X 0,Y 345.559,Z 366.674,A -85,B 0,C 180,E1 -15176.586,E2 -15176.586} C_VEL
LIN {X 0,Y 341.047,Z 481.661,A -85,B 0,C 180,E1 -15179.164,E2 -15179.164} C_VEL
LIN {X 0,Y 339.735,Z 497.153,A -85,B 0,C 180,E1 -15179.72,E2 -15179.72} C_VEL
LIN {X 0,Y 337.967,Z 512.146,A -85,B 0,C 180,E1 -15180.491,E2 -15180.491} C_VEL
LIN {X 0,Y 336.016,Z 526.577,A -85,B 0,C 180,E1 -15181.494,E2 -15181.494} C_VEL
LIN {X 0,Y 333.683,Z 540.667,A -85,B 0,C 180,E1 -15182.737,E2 -15182.737} C_VEL
LIN {X 0,Y 331.228,Z 554.079,A -85,B 0,C 180,E1 -15184.218,E2 -15184.218} C_VEL
LIN {X 0,Y 328.68,Z 566.331,A -85,B 0,C 180,E1 -15185.863,E2 -15185.863} C_VEL
LIN {X 0,Y 326.489,Z 576.946,A -85,B 0,C 180,E1 -15187.594,E2 -15187.594} C_VEL
LIN {X 0,Y 324.254,Z 587.748,A -85,B 0,C 180,E1 -15189.71,E2 -15189.71} C_VEL
LIN {X 0,Y 322.435,Z 595.721,A -85,B 0,C 180,E1 -15191.577,E2 -15191.577} C_VEL
LIN {X 0,Y 320.818,Z 603.624,A -85,B 0,C 180,E1 -15193.782,E2 -15193.782} C_VEL
LIN {X 0,Y 319.621,Z 610.206,A -85,B 0,C 180,E1 -15196.004,E2 -15196.004} C_VEL
LIN {X 0,Y 318.609,Z 616.271,A -85,B 0,C 180,E1 -15198.55,E2 -15198.55} C_VEL
LIN {X 0,Y 318.08,Z 620.961,A -85,B 0,C 180,E1 -15201.103,E2 -15201.103} C_VEL
LIN {X 0,Y 317.799,Z 624.338,A -85,B 0,C 180,E1 -15203.652,E2 -15203.652} C_VEL
LIN {X 0,Y 317.753,Z 626.502,A -85,B 0,C 180,E1 -15206.196,E2 -15206.196} C_VEL
LIN {X 0,Y 317.742,Z 627.497,A -85,B 0,C 180,E1 -15208.733,E2 -15208.733} C_VEL
LIN {X 0,Y 317.743,Z 627.337,A -85,B 0,C 180,E1 -15211.268,E2 -15211.268} C_VEL
LIN {X 0,Y 317.761,Z 626.005,A -85,B 0,C 180,E1 -15213.805,E2 -15213.805} C_VEL
LIN {X 0,Y 317.816,Z 623.428,A -85,B 0,C 180,E1 -15216.348,E2 -15216.348} C_VEL
LIN {X 0,Y 318.078,Z 619.593,A -85,B 0,C 180,E1 -15218.898,E2 -15218.898} C_VEL
LIN {X 0,Y 318.58,Z 614.411,A -85,B 0,C 180,E1 -15221.452,E2 -15221.452} C_VEL
LIN {X 0,Y 319.532,Z 607.752,A -85,B 0,C 180,E1 -15224.001,E2 -15224.001} C_VEL
LIN {X 0,Y 320.655,Z 600.557,A -85,B 0,C 180,E1 -15226.228,E2 -15226.228} C_VEL
LIN {X 0,Y 322.125,Z 591.893,A -85,B 0,C 180,E1 -15228.443,E2 -15228.443} C_VEL
LIN {X 0,Y 324.188,Z 581.552,A -85,B 0,C 180,E1 -15230.609,E2 -15230.609} C_VEL
LIN {X 0,Y 325.719,Z 572.717,A -85,B 0,C 180,E1 -15232.185,E2 -15232.185} C_VEL
LIN {X 0,Y 327.683,Z 561.383,A -85,B 0,C 180,E1 -15233.88,E2 -15233.88} C_VEL
LIN {X 0,Y 329.87,Z 549.12,A -85,B 0,C 180,E1 -15235.39,E2 -15235.39} C_VEL
LIN {X 0,Y 331.951,Z 535.784,A -85,B 0,C 180,E1 -15236.737,E2 -15236.737} C_VEL
LIN {X 0,Y 333.895,Z 521.504,A -85,B 0,C 180,E1 -15237.891,E2 -15237.891} C_VEL
LIN {X 0,Y 335.549,Z 506.989,A -85,B 0,C 180,E1 -15238.798,E2 -15238.798} C_VEL
LIN {X 0,Y 336.92,Z 492.028,A -85,B 0,C 180,E1 -15239.482,E2 -15239.482} C_VEL
LIN {X 0,Y 337.861,Z 476.748,A -85,B 0,C 180,E1 -15239.949,E2 -15239.949} C_VEL
LIN {X 0,Y 341.512,Z 365.093,A -85,B 0,C 180,E1 -15242.4,E2 -15242.4} C_VEL
LIN {X 0,Y 338.169,Z 346.498,A -85,B 0,C 180,E1 -15243.196,E2 -15243.196} C_VEL
LIN {X 0,Y 329.241,Z 326.19,A -85,B 0,C 180,E1 -15244.654,E2 -15244.654} C_VEL
LIN {X 0,Y 324.161,Z 315.334,A -85,B 0,C 180,E1 -15245.509,E2 -15245.509} C_VEL
LIN {X 0,Y 321.22,Z 304.239,A -85,B 0,C 180,E1 -15248.538,E2 -15248.538} C_VEL
LIN {X 0,Y 319.515,Z 298.306,A -85,B 0,C 180,E1 -15250.288,E2 -15250.288} C_VEL
LIN {X 0,Y 319.52,Z 298.302,A -85,B 0,C 180,E1 -15253.459,E2 -15253.459} C_VEL
LIN {X 0,Y 319.552,Z 298.3,A -85,B 0,C 180,E1 -15257.014,E2 -15257.014} C_VEL
LIN {X 0,Y 319.517,Z 298.302,A -85,B 0,C 180,E1 -15260.365,E2 -15260.365} C_VEL
LIN {X 0,Y 319.579,Z 298.296,A -85,B 0,C 180,E1 -15264.456,E2 -15264.456} C_VEL
LIN {X 0,Y 319.525,Z 298.31,A -85,B 0,C 180,E1 -15268.136,E2 -15268.136} C_VEL
LIN {X 0,Y 319.564,Z 298.306,A -85,B 0,C 180,E1 -15271.605,E2 -15271.605} C_VEL
LIN {X 0,Y 319.527,Z 298.312,A -85,B 0,C 180,E1 -15275.296,E2 -15275.296} C_VEL
LIN {X 0,Y 319.564,Z 298.31,A -85,B 0,C 180,E1 -15278.044,E2 -15278.044} C_VEL
LIN {X 0,Y 319.613,Z 298.303,A -85,B 0,C 180,E1 -15282.069,E2 -15282.069} C_VEL
LIN {X 0,Y 319.728,Z 298.259,A -85,B 0,C 180,E1 -15286.006,E2 -15286.006} C_VEL
LIN {X 0,Y 319.73,Z 298.271,A -85,B 0,C 180,E1 -15289.87,E2 -15289.87} C_VEL
LIN {X 0,Y 319.892,Z 298.257,A -85,B 0,C 180,E1 -15293.691,E2 -15293.691} C_VEL
LIN {X 0,Y 320.002,Z 298.233,A -85,B 0,C 180,E1 -15298.739,E2 -15298.739} C_VEL
LIN {X 0,Y 319.95,Z 298.252,A -85,B 0,C 180,E1 -15302.516,E2 -15302.516} C_VEL
LIN {X 0,Y 319.857,Z 298.229,A -85,B 0,C 180,E1 -15306.421,E2 -15306.421} C_VEL
LIN {X 0,Y 319.772,Z 298.261,A -85,B 0,C 180,E1 -15308.848,E2 -15308.848} C_VEL
LIN {X 0,Y 319.671,Z 298.288,A -85,B 0,C 180,E1 -15312.698,E2 -15312.698} C_VEL
LIN {X 0,Y 319.671,Z 298.265,A -85,B 0,C 180,E1 -15315.294,E2 -15315.294} C_VEL
LIN {X 0,Y 319.62,Z 298.279,A -85,B 0,C 180,E1 -15319.256,E2 -15319.256} C_VEL
LIN {X 0,Y 319.532,Z 298.304,A -85,B 0,C 180,E1 -15323.32,E2 -15323.32} C_VEL
LIN {X 0,Y 319.539,Z 298.279,A -85,B 0,C 180,E1 -15326.094,E2 -15326.094} C_VEL
LIN {X 0,Y 319.513,Z 298.289,A -85,B 0,C 180,E1 -15328.938,E2 -15328.938} C_VEL
LIN {X 0,Y 319.513,Z 298.309,A -85,B 0,C 180,E1 -15331.861,E2 -15331.861} C_VEL
LIN {X 0,Y 319.566,Z 298.279,A -85,B 0,C 180,E1 -15335.54,E2 -15335.54} C_VEL
LIN {X 0,Y 319.516,Z 298.308,A -85,B 0,C 180,E1 -15339.66,E2 -15339.66} C_VEL
LIN {X 0,Y 319.506,Z 298.3,A -85,B 0,C 180,E1 -15343.458,E2 -15343.458} C_VEL
LIN {X 0,Y 319.539,Z 298.294,A -85,B 0,C 180,E1 -15347.015,E2 -15347.015} C_VEL
LIN {X 0,Y 319.533,Z 298.309,A -85,B 0,C 180,E1 -15350.369,E2 -15350.369} C_VEL
LIN {X 0,Y 319.564,Z 298.294,A -85,B 0,C 180,E1 -15354.456,E2 -15354.456} C_VEL
LIN {X 0,Y 319.51,Z 298.306,A -85,B 0,C 180,E1 -15358.136,E2 -15358.136} C_VEL
LIN {X 0,Y 319.595,Z 298.299,A -85,B 0,C 180,E1 -15361.589,E2 -15361.589} C_VEL
LIN {X 0,Y 319.587,Z 298.29,A -85,B 0,C 180,E1 -15365.303,E2 -15365.303} C_VEL
LIN {X 0,Y 319.586,Z 298.292,A -85,B 0,C 180,E1 -15369.399,E2 -15369.399} C_VEL
LIN {X 0,Y 319.642,Z 298.296,A -85,B 0,C 180,E1 -15372.072,E2 -15372.072} C_VEL
LIN {X 0,Y 319.717,Z 298.282,A -85,B 0,C 180,E1 -15376.007,E2 -15376.007} C_VEL
LIN {X 0,Y 319.742,Z 298.276,A -85,B 0,C 180,E1 -15379.872,E2 -15379.872} C_VEL
LIN {X 0,Y 319.916,Z 298.261,A -85,B 0,C 180,E1 -15383.377,E2 -15383.377} C_VEL
LIN {X 0,Y 319.947,Z 298.296,A -85,B 0,C 180,E1 -15383.694,E2 -15383.694} C_VEL
LIN {X 0,Y 320.285,Z 299.873,A -85,B 0,C 180,E1 -15384.125,E2 -15384.125} C_VEL
LIN {X 0,Y 327.809,Z 314.66,A -85,B 0,C 180,E1 -15385.38,E2 -15385.38} C_VEL
LIN {X 0,Y 334.983,Z 329.497,A -85,B 0,C 180,E1 -15386.536,E2 -15386.536} C_VEL
LIN {X 0,Y 341.859,Z 345.876,A -85,B 0,C 180,E1 -15387.643,E2 -15387.643} C_VEL
LIN {X 0,Y 338.746,Z 441.947,A -85,B 0,C 180,E1 -15389.747,E2 -15389.747} C_VEL
LIN {X 0,Y 337.818,Z 466.728,A -85,B 0,C 180,E1 -15390.34,E2 -15390.34} C_VEL
LIN {X 0,Y 336.709,Z 482.163,A -85,B 0,C 180,E1 -15390.935,E2 -15390.935} C_VEL
LIN {X 0,Y 335.389,Z 496.567,A -85,B 0,C 180,E1 -15391.726,E2 -15391.726} C_VEL
LIN {X 0,Y 333.801,Z 510.377,A -85,B 0,C 180,E1 -15392.715,E2 -15392.715} C_VEL
LIN {X 0,Y 331.797,Z 524.721,A -85,B 0,C 180,E1 -15394.017,E2 -15394.017} C_VEL
LIN {X 0,Y 329.698,Z 537.911,A -85,B 0,C 180,E1 -15395.504,E2 -15395.504} C_VEL
LIN {X 0,Y 327.531,Z 550.466,A -85,B 0,C 180,E1 -15397.241,E2 -15397.241} C_VEL
LIN {X 0,Y 325.618,Z 561.031,A -85,B 0,C 180,E1 -15399.002,E2 -15399.002} C_VEL
LIN {X 0,Y 323.792,Z 570.802,A -85,B 0,C 180,E1 -15400.947,E2 -15400.947} C_VEL
LIN {X 0,Y 321.952,Z 580.342,A -85,B 0,C 180,E1 -15403.25,E2 -15403.25} C_VEL
LIN {X 0,Y 320.643,Z 587.474,A -85,B 0,C 180,E1 -15405.344,E2 -15405.344} C_VEL
LIN {X 0,Y 319.461,Z 594.676,A -85,B 0,C 180,E1 -15407.937,E2 -15407.937} C_VEL
LIN {X 0,Y 318.588,Z 600.547,A -85,B 0,C 180,E1 -15410.667,E2 -15410.667} C_VEL
LIN {X 0,Y 318.007,Z 604.902,A -85,B 0,C 180,E1 -15413.44,E2 -15413.44} C_VEL
LIN {X 0,Y 317.766,Z 606.637,A -85,B 0,C 180,E1 -15414.942,E2 -15414.942} C_VEL
LIN {X 0,Y 317.489,Z 608.745,A -85,B 0,C 180,E1 -15417.7,E2 -15417.7} C_VEL
LIN {X 0,Y 317.454,Z 609.465,A -85,B 0,C 180,E1 -15420.305,E2 -15420.305} C_VEL
LIN {X 0,Y 317.582,Z 609.028,A -85,B 0,C 180,E1 -15422.767,E2 -15422.767} C_VEL
LIN {X 0,Y 317.8,Z 607.654,A -85,B 0,C 180,E1 -15425.097,E2 -15425.097} C_VEL
LIN {X 0,Y 318.173,Z 605.416,A -85,B 0,C 180,E1 -15427.332,E2 -15427.332} C_VEL
LIN {X 0,Y 318.782,Z 601.912,A -85,B 0,C 180,E1 -15429.741,E2 -15429.741} C_VEL
LIN {X 0,Y 319.688,Z 597.169,A -85,B 0,C 180,E1 -15432.194,E2 -15432.194} C_VEL
LIN {X 0,Y 320.714,Z 592.042,A -85,B 0,C 180,E1 -15434.304,E2 -15434.304} C_VEL
LIN {X 0,Y 320.604,Z 589.517,A -85,B 0,C 180,E1 -15435.256,E2 -15435.256} C_VEL
LIN {X 0,Y 317.366,Z 581.564,A -85,B 0,C 180,E1 -15438.068,E2 -15438.068} C_VEL
LIN {X 0,Y 317.109,Z 578.459,A -85,B 0,C 180,E1 -15438.979,E2 -15438.979} C_VEL
LIN {X 0,Y 317.291,Z 577.353,A -85,B 0,C 180,E1 -15439.274,E2 -15439.274} C_VEL
LIN {X 0,Y 319.418,Z 568.342,A -85,B 0,C 180,E1 -15441.358,E2 -15441.358} C_VEL
LIN {X 0,Y 321.872,Z 557.893,A -85,B 0,C 180,E1 -15443.36,E2 -15443.36} C_VEL
LIN {X 0,Y 324.33,Z 546.51,A -85,B 0,C 180,E1 -15445.169,E2 -15445.169} C_VEL
LIN {X 0,Y 326.845,Z 534.249,A -85,B 0,C 180,E1 -15446.77,E2 -15446.77} C_VEL
LIN {X 0,Y 329.097,Z 521.731,A -85,B 0,C 180,E1 -15448.117,E2 -15448.117} C_VEL
LIN {X 0,Y 331.216,Z 508.259,A -85,B 0,C 180,E1 -15449.292,E2 -15449.292} C_VEL
LIN {X 0,Y 333.174,Z 493.316,A -85,B 0,C 180,E1 -15450.307,E2 -15450.307} C_VEL
LIN {X 0,Y 334.683,Z 478.698,A -85,B 0,C 180,E1 -15451.046,E2 -15451.046} C_VEL
LIN {X 0,Y 335.792,Z 463.289,A -85,B 0,C 180,E1 -15451.581,E2 -15451.581} C_VEL
LIN {X 0,Y 340.299,Z 351.055,A -85,B 0,C 180,E1 -15454.141,E2 -15454.141} C_VEL
LIN {X 0,Y 333.286,Z 335.832,A -85,B 0,C 180,E1 -15455.536,E2 -15455.536} C_VEL
LIN {X 0,Y 326.193,Z 322.636,A -85,B 0,C 180,E1 -15456.987,E2 -15456.987} C_VEL
LIN {X 0,Y 318.493,Z 309.899,A -85,B 0,C 180,E1 -15458.651,E2 -15458.651} C_VEL
LIN {X 0,Y 315.482,Z 305.379,A -85,B 0,C 180,E1 -15459.326,E2 -15459.326} C_VEL
LIN {X 0,Y 313.384,Z 301.757,A -85,B 0,C 180,E1 -15459.833,E2 -15459.833} C_VEL
LIN {X 0,Y 312.638,Z 299.16,A -85,B 0,C 180,E1 -15460.931,E2 -15460.931} C_VEL
LIN {X 0,Y 312.688,Z 299.16,A -85,B 0,C 180,E1 -15465.115,E2 -15465.115} C_VEL
LIN {X 0,Y 312.687,Z 299.159,A -85,B 0,C 180,E1 -15469.644,E2 -15469.644} C_VEL
LIN {X 0,Y 312.842,Z 299.14,A -85,B 0,C 180,E1 -15472.256,E2 -15472.256} C_VEL
LIN {X 0,Y 312.703,Z 299.158,A -85,B 0,C 180,E1 -15474.844,E2 -15474.844} C_VEL
LIN {X 0,Y 312.98,Z 299.121,A -85,B 0,C 180,E1 -15478.715,E2 -15478.715} C_VEL
LIN {X 0,Y 312.98,Z 299.12,A -85,B 0,C 180,E1 -15481.289,E2 -15481.289} C_VEL
LIN {X 0,Y 312.694,Z 299.155,A -85,B 0,C 180,E1 -15485.16,E2 -15485.16} C_VEL
LIN {X 0,Y 312.81,Z 299.138,A -85,B 0,C 180,E1 -15487.749,E2 -15487.749} C_VEL
LIN {X 0,Y 312.655,Z 299.161,A -85,B 0,C 180,E1 -15491.674,E2 -15491.674} C_VEL
LIN {X 0,Y 312.661,Z 299.161,A -85,B 0,C 180,E1 -15494.867,E2 -15494.867} C_VEL
LIN {X 0,Y 312.542,Z 299.176,A -85,B 0,C 180,E1 -15499.195,E2 -15499.195} C_VEL
LIN {X 0,Y 312.512,Z 299.177,A -85,B 0,C 180,E1 -15502.779,E2 -15502.779} C_VEL
LIN {X 0,Y 312.481,Z 299.182,A -85,B 0,C 180,E1 -15506.734,E2 -15506.734} C_VEL
LIN {X 0,Y 312.463,Z 299.184,A -85,B 0,C 180,E1 -15509.66,E2 -15509.66} C_VEL
LIN {X 0,Y 312.516,Z 299.177,A -85,B 0,C 180,E1 -15513.691,E2 -15513.691} C_VEL
LIN {X 0,Y 312.506,Z 299.179,A -85,B 0,C 180,E1 -15517.39,E2 -15517.39} C_VEL
LIN {X 0,Y 312.437,Z 299.19,A -85,B 0,C 180,E1 -15520.719,E2 -15520.719} C_VEL
LIN {X 0,Y 312.448,Z 299.189,A -85,B 0,C 180,E1 -15524.212,E2 -15524.212} C_VEL
LIN {X 0,Y 312.449,Z 299.259,A -85,B 0,C 180,E1 -15525.742,E2 -15525.742} C_VEL
LIN {X 0,Y 315.531,Z 308.724,A -85,B 0,C 180,E1 -15529.229,E2 -15529.229} C_VEL
LIN {X 0,Y 317.111,Z 313.7,A -85,B 0,C 180,E1 -15530.87,E2 -15530.87} C_VEL
LIN {X 0,Y 325.412,Z 328.305,A -85,B 0,C 180,E1 -15532.7,E2 -15532.7} C_VEL
LIN {X 0,Y 332.171,Z 341.823,A -85,B 0,C 180,E1 -15534.115,E2 -15534.115} C_VEL
LIN {X 0,Y 337.667,Z 354.047,A -85,B 0,C 180,E1 -15535.231,E2 -15535.231} C_VEL
LIN {X 0,Y 339.802,Z 366.823,A -85,B 0,C 180,E1 -15535.868,E2 -15535.868} C_VEL
LIN {X 0,Y 336.222,Z 457.669,A -85,B 0,C 180,E1 -15537.924,E2 -15537.924} C_VEL
LIN {X 0,Y 335.034,Z 483.251,A -85,B 0,C 180,E1 -15538.548,E2 -15538.548} C_VEL
LIN {X 0,Y 333.617,Z 498.858,A -85,B 0,C 180,E1 -15539.149,E2 -15539.149} C_VEL
LIN {X 0,Y 331.703,Z 513.887,A -85,B 0,C 180,E1 -15539.964,E2 -15539.964} C_VEL
LIN {X 0,Y 329.538,Z 528.589,A -85,B 0,C 180,E1 -15541.039,E2 -15541.039} C_VEL
LIN {X 0,Y 327.128,Z 542.39,A -85,B 0,C 180,E1 -15542.318,E2 -15542.318} C_VEL
LIN {X 0,Y 324.589,Z 555.466,A -85,B 0,C 180,E1 -15543.823,E2 -15543.823} C_VEL
LIN {X 0,Y 321.966,Z 567.456,A -85,B 0,C 180,E1 -15545.498,E2 -15545.498} C_VEL
LIN {X 0,Y 319.575,Z 578.518,A -85,B 0,C 180,E1 -15547.38,E2 -15547.38} C_VEL
LIN {X 0,Y 317.216,Z 589.173,A -85,B 0,C 180,E1 -15549.578,E2 -15549.578} C_VEL
LIN {X 0,Y 315.387,Z 596.954,A -85,B 0,C 180,E1 -15551.487,E2 -15551.487} C_VEL
LIN {X 0,Y 313.701,Z 604.595,A -85,B 0,C 180,E1 -15553.738,E2 -15553.738} C_VEL
LIN {X 0,Y 312.358,Z 611.764,A -85,B 0,C 180,E1 -15556.336,E2 -15556.336} C_VEL
LIN {X 0,Y 311.391,Z 617.431,A -85,B 0,C 180,E1 -15558.94,E2 -15558.94} C_VEL
LIN {X 0,Y 311.005,Z 620.831,A -85,B 0,C 180,E1 -15560.899,E2 -15560.899} C_VEL
LIN {X 0,Y 310.708,Z 624.19,A -85,B 0,C 180,E1 -15563.507,E2 -15563.507} C_VEL
LIN {X 0,Y 310.664,Z 626.327,A -85,B 0,C 180,E1 -15566.109,E2 -15566.109} C_VEL
LIN {X 0,Y 310.656,Z 627.299,A -85,B 0,C 180,E1 -15568.704,E2 -15568.704} C_VEL
LIN {X 0,Y 310.657,Z 627.116,A -85,B 0,C 180,E1 -15571.297,E2 -15571.297} C_VEL
LIN {X 0,Y 310.674,Z 625.763,A -85,B 0,C 180,E1 -15573.892,E2 -15573.892} C_VEL
LIN {X 0,Y 310.723,Z 623.17,A -85,B 0,C 180,E1 -15576.494,E2 -15576.494} C_VEL
LIN {X 0,Y 311.003,Z 619.307,A -85,B 0,C 180,E1 -15579.102,E2 -15579.102} C_VEL
LIN {X 0,Y 311.575,Z 614.093,A -85,B 0,C 180,E1 -15581.713,E2 -15581.713} C_VEL
LIN {X 0,Y 312.527,Z 607.393,A -85,B 0,C 180,E1 -15584.322,E2 -15584.322} C_VEL
LIN {X 0,Y 313.75,Z 600.156,A -85,B 0,C 180,E1 -15586.595,E2 -15586.595} C_VEL
LIN {X 0,Y 315.309,Z 591.44,A -85,B 0,C 180,E1 -15588.856,E2 -15588.856} C_VEL
LIN {X 0,Y 317.396,Z 581.249,A -85,B 0,C 180,E1 -15591.027,E2 -15591.027} C_VEL
LIN {X 0,Y 319.07,Z 572.142,A -85,B 0,C 180,E1 -15592.673,E2 -15592.673} C_VEL
LIN {X 0,Y 321.161,Z 560.76,A -85,B 0,C 180,E1 -15594.396,E2 -15594.396} C_VEL
LIN {X 0,Y 323.407,Z 548.406,A -85,B 0,C 180,E1 -15595.934,E2 -15595.934} C_VEL
LIN {X 0,Y 325.559,Z 535.076,A -85,B 0,C 180,E1 -15597.292,E2 -15597.292} C_VEL
LIN {X 0,Y 327.563,Z 520.514,A -85,B 0,C 180,E1 -15598.479,E2 -15598.479} C_VEL
LIN {X 0,Y 329.307,Z 505.769,A -85,B 0,C 180,E1 -15599.397,E2 -15599.397} C_VEL
LIN {X 0,Y 330.729,Z 490.411,A -85,B 0,C 180,E1 -15600.09,E2 -15600.09} C_VEL
LIN {X 0,Y 331.676,Z 474.25,A -85,B 0,C 180,E1 -15600.567,E2 -15600.567} C_VEL
LIN {X 0,Y 335.352,Z 366.189,A -85,B 0,C 180,E1 -15602.97,E2 -15602.97} C_VEL
LIN {X 0,Y 332.392,Z 349.413,A -85,B 0,C 180,E1 -15603.706,E2 -15603.706} C_VEL
LIN {X 0,Y 324.055,Z 330.249,A -85,B 0,C 180,E1 -15605.11,E2 -15605.11} C_VEL
LIN {X 0,Y 316.903,Z 315.076,A -85,B 0,C 180,E1 -15606.359,E2 -15606.359} C_VEL
LIN {X 0,Y 313.835,Z 304.088,A -85,B 0,C 180,E1 -15609.482,E2 -15609.482} C_VEL
LIN {X 0,Y 312.459,Z 299.185,A -85,B 0,C 180,E1 -15610.965,E2 -15610.965} C_VEL
LIN {X 0,Y 312.452,Z 299.186,A -85,B 0,C 180,E1 -15614.209,E2 -15614.209} C_VEL
LIN {X 0,Y 312.455,Z 299.192,A -85,B 0,C 180,E1 -15617.924,E2 -15617.924} C_VEL
LIN {X 0,Y 312.477,Z 299.186,A -85,B 0,C 180,E1 -15621.923,E2 -15621.923} C_VEL
LIN {X 0,Y 312.531,Z 299.176,A -85,B 0,C 180,E1 -15624.218,E2 -15624.218} C_VEL
LIN {X 0,Y 312.503,Z 299.18,A -85,B 0,C 180,E1 -15627.332,E2 -15627.332} C_VEL
LIN {X 0,Y 312.494,Z 299.185,A -85,B 0,C 180,E1 -15631.294,E2 -15631.294} C_VEL
LIN {X 0,Y 312.517,Z 299.184,A -85,B 0,C 180,E1 -15634.703,E2 -15634.703} C_VEL
LIN {X 0,Y 312.538,Z 299.18,A -85,B 0,C 180,E1 -15637.523,E2 -15637.523} C_VEL
LIN {X 0,Y 312.566,Z 299.177,A -85,B 0,C 180,E1 -15641.65,E2 -15641.65} C_VEL
LIN {X 0,Y 312.683,Z 299.139,A -85,B 0,C 180,E1 -15645.684,E2 -15645.684} C_VEL
LIN {X 0,Y 312.68,Z 299.145,A -85,B 0,C 180,E1 -15649.639,E2 -15649.639} C_VEL
LIN {X 0,Y 312.834,Z 299.137,A -85,B 0,C 180,E1 -15653.548,E2 -15653.548} C_VEL
LIN {X 0,Y 312.969,Z 299.109,A -85,B 0,C 180,E1 -15658.711,E2 -15658.711} C_VEL
LIN {X 0,Y 312.899,Z 299.131,A -85,B 0,C 180,E1 -15662.573,E2 -15662.573} C_VEL
LIN {X 0,Y 312.812,Z 299.106,A -85,B 0,C 180,E1 -15666.448,E2 -15666.448} C_VEL
LIN {X 0,Y 312.723,Z 299.14,A -85,B 0,C 180,E1 -15669.049,E2 -15669.049} C_VEL
LIN {X 0,Y 312.625,Z 299.168,A -85,B 0,C 180,E1 -15672.989,E2 -15672.989} C_VEL
LIN {X 0,Y 312.613,Z 299.139,A -85,B 0,C 180,E1 -15675.649,E2 -15675.649} C_VEL
LIN {X 0,Y 312.55,Z 299.165,A -85,B 0,C 180,E1 -15679.709,E2 -15679.709} C_VEL
LIN {X 0,Y 312.508,Z 299.182,A -85,B 0,C 180,E1 -15682.774,E2 -15682.774} C_VEL
LIN {X 0,Y 312.471,Z 299.152,A -85,B 0,C 180,E1 -15686.73,E2 -15686.73} C_VEL
LIN {X 0,Y 312.458,Z 299.176,A -85,B 0,C 180,E1 -15689.656,E2 -15689.656} C_VEL
LIN {X 0,Y 312.508,Z 299.176,A -85,B 0,C 180,E1 -15693.687,E2 -15693.687} C_VEL
LIN {X 0,Y 312.497,Z 299.155,A -85,B 0,C 180,E1 -15697.386,E2 -15697.386} C_VEL
LIN {X 0,Y 312.428,Z 299.192,A -85,B 0,C 180,E1 -15700.715,E2 -15700.715} C_VEL
LIN {X 0,Y 312.437,Z 299.174,A -85,B 0,C 180,E1 -15704.208,E2 -15704.208} C_VEL
LIN {X 0,Y 312.47,Z 299.186,A -85,B 0,C 180,E1 -15707.917,E2 -15707.917} C_VEL
LIN {X 0,Y 312.484,Z 299.181,A -85,B 0,C 180,E1 -15710.969,E2 -15710.969} C_VEL
LIN {X 0,Y 312.517,Z 299.17,A -85,B 0,C 180,E1 -15714.219,E2 -15714.219} C_VEL
LIN {X 0,Y 312.487,Z 299.183,A -85,B 0,C 180,E1 -15717.332,E2 -15717.332} C_VEL
LIN {X 0,Y 312.554,Z 299.175,A -85,B 0,C 180,E1 -15721.823,E2 -15721.823} C_VEL
LIN {X 0,Y 312.569,Z 299.164,A -85,B 0,C 180,E1 -15724.71,E2 -15724.71} C_VEL
LIN {X 0,Y 312.521,Z 299.174,A -85,B 0,C 180,E1 -15728.911,E2 -15728.911} C_VEL
LIN {X 0,Y 312.622,Z 299.17,A -85,B 0,C 180,E1 -15731.655,E2 -15731.655} C_VEL
LIN {X 0,Y 312.678,Z 299.161,A -85,B 0,C 180,E1 -15735.685,E2 -15735.685} C_VEL
LIN {X 0,Y 312.687,Z 299.155,A -85,B 0,C 180,E1 -15739.641,E2 -15739.641} C_VEL
LIN {X 0,Y 312.888,Z 299.306,A -85,B 0,C 180,E1 -15743.065,E2 -15743.065} C_VEL
LIN {X 0,Y 313.075,Z 300.106,A -85,B 0,C 180,E1 -15743.272,E2 -15743.272} C_VEL
LIN {X 0,Y 314.654,Z 303.143,A -85,B 0,C 180,E1 -15743.551,E2 -15743.551} C_VEL
LIN {X 0,Y 325.617,Z 324.685,A -85,B 0,C 180,E1 -15745.408,E2 -15745.408} C_VEL
LIN {X 0,Y 332.546,Z 340.013,A -85,B 0,C 180,E1 -15746.559,E2 -15746.559} C_VEL
LIN {X 0,Y 335.759,Z 348.285,A -85,B 0,C 180,E1 -15747.102,E2 -15747.102} C_VEL
LIN {X 0,Y 331.659,Z 464.193,A -85,B 0,C 180,E1 -15749.696,E2 -15749.696} C_VEL
LIN {X 0,Y 330.578,Z 480.078,A -85,B 0,C 180,E1 -15750.279,E2 -15750.279} C_VEL
LIN {X 0,Y 329.175,Z 495.357,A -85,B 0,C 180,E1 -15751.101,E2 -15751.101} C_VEL
LIN {X 0,Y 327.68,Z 508.038,A -85,B 0,C 180,E1 -15751.997,E2 -15751.997} C_VEL
LIN {X 0,Y 325.739,Z 522.154,A -85,B 0,C 180,E1 -15753.246,E2 -15753.246} C_VEL
LIN {X 0,Y 323.831,Z 534.078,A -85,B 0,C 180,E1 -15754.546,E2 -15754.546} C_VEL
LIN {X 0,Y 321.728,Z 546.006,A -85,B 0,C 180,E1 -15756.112,E2 -15756.112} C_VEL
LIN {X 0,Y 319.401,Z 558.249,A -85,B 0,C 180,E1 -15758.065,E2 -15758.065} C_VEL
LIN {X 0,Y 317.301,Z 569.225,A -85,B 0,C 180,E1 -15760.206,E2 -15760.206} C_VEL
LIN {X 0,Y 315.544,Z 578.034,A -85,B 0,C 180,E1 -15762.28,E2 -15762.28} C_VEL
LIN {X 0,Y 314.165,Z 585.073,A -85,B 0,C 180,E1 -15764.244,E2 -15764.244} C_VEL
LIN {X 0,Y 313.046,Z 591.215,A -85,B 0,C 180,E1 -15766.297,E2 -15766.297} C_VEL
LIN {X 0,Y 311.991,Z 597.563,A -85,B 0,C 180,E1 -15768.907,E2 -15768.907} C_VEL
LIN {X 0,Y 311.423,Z 601.858,A -85,B 0,C 180,E1 -15771.165,E2 -15771.165} C_VEL
LIN {X 0,Y 310.793,Z 605.884,A -85,B 0,C 180,E1 -15774.018,E2 -15774.018} C_VEL
LIN {X 0,Y 310.579,Z 607.355,A -85,B 0,C 180,E1 -15775.463,E2 -15775.463} C_VEL
LIN {X 0,Y 310.358,Z 609.219,A -85,B 0,C 180,E1 -15778.393,E2 -15778.393} C_VEL
LIN {X 0,Y 310.353,Z 609.689,A -85,B 0,C 180,E1 -15780.632,E2 -15780.632} C_VEL
LIN {X 0,Y 310.502,Z 609.148,A -85,B 0,C 180,E1 -15783.132,E2 -15783.132} C_VEL
LIN {X 0,Y 310.829,Z 607.239,A -85,B 0,C 180,E1 -15786.005,E2 -15786.005} C_VEL
LIN {X 0,Y 311.182,Z 605.371,A -85,B 0,C 180,E1 -15787.776,E2 -15787.776} C_VEL
LIN {X 0,Y 311.781,Z 602.191,A -85,B 0,C 180,E1 -15789.972,E2 -15789.972} C_VEL
LIN {X 0,Y 312.69,Z 597.651,A -85,B 0,C 180,E1 -15792.396,E2 -15792.396} C_VEL
LIN {X 0,Y 313.957,Z 591.753,A -85,B 0,C 180,E1 -15794.866,E2 -15794.866} C_VEL
LIN {X 0,Y 315.596,Z 584.518,A -85,B 0,C 180,E1 -15797.295,E2 -15797.295} C_VEL
LIN {X 0,Y 317.291,Z 577.353,A -85,B 0,C 180,E1 -15799.274,E2 -15799.274} C_VEL
LIN {X 0,Y 317.459,Z 574.039,A -85,B 0,C 180,E1 -15800.158,E2 -15800.158} C_VEL
LIN {X 0,Y 316.122,Z 568.528,A -85,B 0,C 180,E1 -15801.632,E2 -15801.632} C_VEL
LIN {X 0,Y 314.944,Z 562.601,A -85,B 0,C 180,E1 -15803.054,E2 -15803.054} C_VEL
LIN {X 0,Y 315.34,Z 558.594,A -85,B 0,C 180,E1 -15803.84,E2 -15803.84} C_VEL
LIN {X 0,Y 317.94,Z 547.165,A -85,B 0,C 180,E1 -15805.704,E2 -15805.704} C_VEL
LIN {X 0,Y 320.501,Z 535.318,A -85,B 0,C 180,E1 -15807.295,E2 -15807.295} C_VEL
LIN {X 0,Y 322.917,Z 522.621,A -85,B 0,C 180,E1 -15808.702,E2 -15808.702} C_VEL
LIN {X 0,Y 325.061,Z 509.772,A -85,B 0,C 180,E1 -15809.859,E2 -15809.859} C_VEL
LIN {X 0,Y 326.984,Z 496.007,A -85,B 0,C 180,E1 -15810.844,E2 -15810.844} C_VEL
LIN {X 0,Y 328.638,Z 480.947,A -85,B 0,C 180,E1 -15811.656,E2 -15811.656} C_VEL
LIN {X 0,Y 329.874,Z 465.845,A -85,B 0,C 180,E1 -15812.217,E2 -15812.217} C_VEL
LIN {X 0,Y 334.694,Z 353.457,A -85,B 0,C 180,E1 -15814.823,E2 -15814.823} C_VEL
LIN {X 0,Y 328.322,Z 339.573,A -85,B 0,C 180,E1 -15816.143,E2 -15816.143} C_VEL
LIN {X 0,Y 321.303,Z 326.389,A -85,B 0,C 180,E1 -15817.645,E2 -15817.645} C_VEL
LIN {X 0,Y 314.133,Z 314.434,A -85,B 0,C 180,E1 -15819.259,E2 -15819.259} C_VEL
LIN {X 0,Y 308.765,Z 306.233,A -85,B 0,C 180,E1 -15820.542,E2 -15820.542} C_VEL
LIN {X 0,Y 306.136,Z 301.975,A -85,B 0,C 180,E1 -15821.255,E2 -15821.255} C_VEL
LIN {X 0,Y 305.55,Z 300.051,A -85,B 0,C 180,E1 -15822.086,E2 -15822.086} C_VEL
LIN {X 0,Y 305.637,Z 300.038,A -85,B 0,C 180,E1 -15825.351,E2 -15825.351} C_VEL
LIN {X 0,Y 305.624,Z 300.038,A -85,B 0,C 180,E1 -15829.402,E2 -15829.402} C_VEL
LIN {X 0,Y 305.786,Z 300.018,A -85,B 0,C 180,E1 -15832.076,E2 -15832.076} C_VEL
LIN {X 0,Y 305.675,Z 300.032,A -85,B 0,C 180,E1 -15834.726,E2 -15834.726} C_VEL
LIN {X 0,Y 305.947,Z 299.997,A -85,B 0,C 180,E1 -15838.686,E2 -15838.686} C_VEL
LIN {X 0,Y 305.947,Z 299.996,A -85,B 0,C 180,E1 -15841.318,E2 -15841.318} C_VEL
LIN {X 0,Y 305.663,Z 300.031,A -85,B 0,C 180,E1 -15845.279,E2 -15845.279} C_VEL
LIN {X 0,Y 305.754,Z 300.017,A -85,B 0,C 180,E1 -15847.929,E2 -15847.929} C_VEL
LIN {X 0,Y 305.591,Z 300.042,A -85,B 0,C 180,E1 -15851.948,E2 -15851.948} C_VEL
LIN {X 0,Y 305.602,Z 300.041,A -85,B 0,C 180,E1 -15855.016,E2 -15855.016} C_VEL
LIN {X 0,Y 305.511,Z 300.055,A -85,B 0,C 180,E1 -15858.789,E2 -15858.789} C_VEL
LIN {X 0,Y 305.451,Z 300.055,A -85,B 0,C 180,E1 -15863.028,E2 -15863.028} C_VEL
LIN {X 0,Y 305.448,Z 300.056,A -85,B 0,C 180,E1 -15866.193,E2 -15866.193} C_VEL
LIN {X 0,Y 305.42,Z 300.058,A -85,B 0,C 180,E1 -15869.028,E2 -15869.028} C_VEL
LIN {X 0,Y 305.431,Z 300.057,A -85,B 0,C 180,E1 -15871.956,E2 -15871.956} C_VEL
LIN {X 0,Y 305.457,Z 300.058,A -85,B 0,C 180,E1 -15875.116,E2 -15875.116} C_VEL
LIN {X 0,Y 305.431,Z 300.06,A -85,B 0,C 180,E1 -15878.527,E2 -15878.527} C_VEL
LIN {X 0,Y 305.432,Z 300.066,A -85,B 0,C 180,E1 -15882.583,E2 -15882.583} C_VEL
LIN {X 0,Y 305.434,Z 300.23,A -85,B 0,C 180,E1 -15884.571,E2 -15884.571} C_VEL
LIN {X 0,Y 308.607,Z 309.612,A -85,B 0,C 180,E1 -15888.248,E2 -15888.248} C_VEL
LIN {X 0,Y 309.762,Z 313.396,A -85,B 0,C 180,E1 -15889.533,E2 -15889.533} C_VEL
LIN {X 0,Y 316.63,Z 325.102,A -85,B 0,C 180,E1 -15891.166,E2 -15891.166} C_VEL
LIN {X 0,Y 321.128,Z 333.23,A -85,B 0,C 180,E1 -15892.178,E2 -15892.178} C_VEL
LIN {X 0,Y 327.318,Z 345.733,A -85,B 0,C 180,E1 -15893.528,E2 -15893.528} C_VEL
LIN {X 0,Y 332.45,Z 357.258,A -85,B 0,C 180,E1 -15894.609,E2 -15894.609} C_VEL
LIN {X 0,Y 334.188,Z 368.499,A -85,B 0,C 180,E1 -15895.176,E2 -15895.176} C_VEL
LIN {X 0,Y 329.388,Z 480.563,A -85,B 0,C 180,E1 -15897.765,E2 -15897.765} C_VEL
LIN {X 0,Y 328.002,Z 496.227,A -85,B 0,C 180,E1 -15898.336,E2 -15898.336} C_VEL
LIN {X 0,Y 326.102,Z 511.303,A -85,B 0,C 180,E1 -15899.124,E2 -15899.124} C_VEL
LIN {X 0,Y 323.895,Z 526.146,A -85,B 0,C 180,E1 -15900.18,E2 -15900.18} C_VEL
LIN {X 0,Y 321.418,Z 539.914,A -85,B 0,C 180,E1 -15901.426,E2 -15901.426} C_VEL
LIN {X 0,Y 318.768,Z 553.355,A -85,B 0,C 180,E1 -15902.954,E2 -15902.954} C_VEL
LIN {X 0,Y 315.968,Z 565.639,A -85,B 0,C 180,E1 -15904.65,E2 -15904.65} C_VEL
LIN {X 0,Y 313.345,Z 577.059,A -85,B 0,C 180,E1 -15906.576,E2 -15906.576} C_VEL
LIN {X 0,Y 310.88,Z 587.847,A -85,B 0,C 180,E1 -15908.796,E2 -15908.796} C_VEL
LIN {X 0,Y 308.597,Z 596.976,A -85,B 0,C 180,E1 -15911.064,E2 -15911.064} C_VEL
LIN {X 0,Y 306.849,Z 604.568,A -85,B 0,C 180,E1 -15913.365,E2 -15913.365} C_VEL
LIN {X 0,Y 305.397,Z 611.689,A -85,B 0,C 180,E1 -15916.018,E2 -15916.018} C_VEL
LIN {X 0,Y 304.382,Z 617.324,A -85,B 0,C 180,E1 -15918.682,E2 -15918.682} C_VEL
LIN {X 0,Y 303.954,Z 620.698,A -85,B 0,C 180,E1 -15920.686,E2 -15920.686} C_VEL
LIN {X 0,Y 303.627,Z 624.044,A -85,B 0,C 180,E1 -15923.355,E2 -15923.355} C_VEL
LIN {X 0,Y 303.559,Z 626.155,A -85,B 0,C 180,E1 -15926.018,E2 -15926.018} C_VEL
LIN {X 0,Y 303.572,Z 627.102,A -85,B 0,C 180,E1 -15928.674,E2 -15928.674} C_VEL
LIN {X 0,Y 303.574,Z 626.891,A -85,B 0,C 180,E1 -15931.327,E2 -15931.327} C_VEL
LIN {X 0,Y 303.572,Z 625.509,A -85,B 0,C 180,E1 -15933.983,E2 -15933.983} C_VEL
LIN {X 0,Y 303.638,Z 622.9,A -85,B 0,C 180,E1 -15936.646,E2 -15936.646} C_VEL
LIN {X 0,Y 303.945,Z 619.004,A -85,B 0,C 180,E1 -15939.315,E2 -15939.315} C_VEL
